// SIMATIC S7-200 SMART project (STEP 7-Micro/WIN SMART), CPU ST20

SYMBOL_TABLE USER1
Btn启动气密          M1.0
Btn停止气密          M1.1
i水箱升到位           M1.2
i水箱j降到位          M1.3
iMaual           M1.4
iAutoGas         M1.5
iResetSingle     M1.6
iStop急停          M1.7
iStartSingle     M2.0
i顶缸上限位           M2.1
i顶杆下限位           M2.2
iHas销钉1          M2.3
iHas销钉2          M2.4
iBYLOK           M2.5
iBYLNG           M2.6
Btn清零合格不合格计数     M2.7
Btn顶缸伸出          M3.0
Btn顶缸缩回          M3.1
Q顶缸伸出启停          M3.2
Q顶缸缩回启停          M3.3
iAutoWater       M3.4
Btn侧顶油伸出         M3.5
Btn侧顶油缩回         M3.6
Q侧顶油伸出启停         M3.7
Q侧顶油缩回启停         M4.0
Btn侧气顶出          M4.2
Btn侧气缩回          M4.3
Q侧气顶出            M4.4
Q侧气缩回            M4.5
Btn高压气检启停        M4.7
Btn低压气检启停        M5.0
Q高压气检启停          M5.1
Q低压气检启停          M5.2
Btn打点伸出          M5.4
Btn打点缩回          M5.5
Q打点伸出            M5.6
Q打点缩回            M5.7
Btn水箱上升启停        M6.1
Btn水箱下降启停        M6.2
Q水箱上升启停          M6.3
Q水箱下降启停          M6.4
Btn高压水检启停        M6.6
Q高压水检启停          M6.7
Btn低压水检启停        M7.0
Q低压水检启停          M7.1
i光栅              M7.3
Btn工作台退回         M7.4
Q工作台推出           M7.5
Q工作台退回           M7.6
Q启动气密仪           M7.7
Q停止气密仪           M8.0
QOK              M8.1
QNG              M8.2
QError报警         M8.3
Q启动运行灯           M8.4
Q三色绿运行           M8.5
Q三色红故障           M8.6
Q三色黄等待           M8.7
Q24V照明灯          M9.0
Q原位指示            M9.1
UISetEnable侧油    M9.3
UISetEnable侧气    M9.4
UISetEnable水箱    M9.5
UISetEnable高压水气检 M9.6
UISetEnable低压水气检 M9.7
UISetEnablee一切换二路 M10.0
MaualVirtual启停气密仪 M10.1
UISetEnable1     M10.2
UIBtnExecute1    M10.3
UISinaPosDone1   M10.4
UISetEnable2     M10.5
UIBtnExecute2    M10.6
UISinaPosDone2   M10.7
UISetEnable销钉    M11.0
CondTrue水箱上升     M11.1
CondTrue水箱下降     M11.2
CondTrue打点伸      M11.3
CondTrue打点缩      M11.4
CondTrueJOG启动气密  M11.5
CondTrueJOG停止气密  M11.6
CondTrue侧气伸      M11.7
CondTrue侧气缩      M12.0
CondTrue一路水检     M12.1
CondTrue二路水检     M12.2
CondTrue有码       M12.3
CondTrue气检合格     M12.4
CondTrue气检不合格    M12.5
CondTrue水检合格     M12.6
CondTrue水检不合格    M12.7
CondTrue工作台推出    M13.0
CondTrue工作台缩回    M13.1
CondTrue顶缸伸      M13.2
CondTrue顶缸缩      M13.3
CondTrue侧油伸      M13.4
CondTrue侧油缩      M13.5
CondTrue一路气检启停   M13.6
CondTrue二路气检启停   M13.7
CondTrue启停气密仪    M14.0
Device当前气密仪状态    M14.1
CondTrue三路气检启停   M14.2
CondTrue关机       M14.3
CondTrueUI气检采集   M14.4
CondTrueUI水检采集   M14.5
UISetEnable扫码枪   M14.6
UIWarning警告      M14.7
UISetSwitch福田    M15.0
CondTrue自锁延迟     M15.1
QLogic伺服启动1      M15.2
QLogic伺服启动2      M15.3
CondTrue伺服启动1    M15.4
CondTrue伺服启动2    M15.5
UIBtnDog上升1      M15.6
UIBtnDog下降1      M15.7
IError泵1         M16.0
IError泵2         M16.1
RunSeq           VW22
UIRunMode        VW28
CountGasRun合格    VW100
CountGasRun不合格   VW102
CountGasRun总数    VW104
RTU扭力1           VW106
RTU扭力2           VW108
UISet无操作待机       VW116
sys待机分钟          VW118
UISet延时复位        VW120
Logic延时复位计时      VW122
UISet福田延时检测      VW124
Logic福田延时计数      VW126
UISetNG福田延时检测    VW128
LogicNG福田延时计数    VW130
UIConv扭力1        VD132
UIConv扭力2        VD136
UISet扭力OK下限1     VD140
UISet扭力OK上限1     VD144
UISet扭力OK下限2     VD148
UISet扭力OK上限2     VD152
UISet伺服距离OK下限1   VD156
UISet伺服距离OK上限1   VD160
UISet伺服距离OK下限2   VD164
UISet伺服距离OK上限2   VD168
UIData扫码枪数据1     VW180
UIData扫码枪数据2     VW182
UIData扫码枪数据3     VW184
UIData扫码枪数据4     VW186
UIData扫码枪数据5     VW188
UIData扫码枪数据6     VW190
UIData扫码枪数据7     VW192
UIData扫码枪数据8     VW194
UIData扫码枪数据9     VW196
UIData扫码枪数据10    VW198
UIData扫码枪数据11    VW200
UIData扫码枪数据12    VW202
UIData扫码枪数据13    VW204
UIData扫码枪数据14    VW206
UIData扫码枪数据15    VW208
UIData扫码枪数据16    VW210
UIData扫码枪数据17    VW212
UIData扫码枪数据18    VW214
UIData扫码枪数据19    VW216
UIData扫码枪数据20    VW218
UIData扫码枪数据21    VW220
UIData扫码枪数据22    VW222
UIData扫码枪数据23    VW224
UIData扫码枪数据24    VW226
UIData扫码枪数据25    VW228
UIData扫码枪数据26    VW230
UIData扫码枪数据27    VW232
UIData扫码枪数据28    VW234
UIData扫码枪数据29    VW236
UIData扫码枪数据30    VW238
UIData扫码枪数据31    VW240
UIData扫码枪数据32    VW242
UIData扫码枪数据33    VW244
UIData扫码枪数据34    VW246
UIData扫码枪数据35    VW248
UIData扫码枪数据36    VW250
UIData扫码枪数据37    VW252
UIData扫码枪数据38    VW254
UIData扫码枪数据39    VW256
UIData扫码枪数据40    VW258
Map气检合格不合格       VW260
UI操作员1           VW262
UI操作员2           VW264
UI操作员3           VW266
UI操作员4           VW268
UI操作员5           VW270
UI操作员6           VW272
UI操作员7           VW274
UI操作员8           VW276
UI操作员9           VW278
UI操作员10          VW280
UI压力值1           VD282
UI扭压力判定结果1       VW286
UI伸出距离1          VD288
UI伸出距离判定1        VW292
UI压力值2           VD294
UI扭压力判定结果2       VW298
UI伸出距离2          VD300
UI伸出距离判定2        VW304
UISetServeMode1  VW500
UISetServePos1   VD502
UISetMDI1        VD506
UISetServeMode2  VW510
UISetServePos2   VD512
UISetMDI2        VD516
UISetZeroOffset1 VD520
UISetZeroOffset2 VD524
Positive1        V600.0
Negative1        V600.1
UISetJodForward1 V600.2
UISetJodReserve1 V600.3
UIBtnFlyRef1     V600.4   // 其他模式下回零
UISetResetErr1   V600.5
UISetOverV1      VW602    // 速度倍率（控制旋转快慢）
UISetOverAcc1    VW604    // 加速倍率（控制启动快慢）
UISetOverDec1    VW606    // 减速度倍率（控制停止快慢）
ConfigEpos1      VD608
ActPosition1     VD612
Axisenabled1     V650.0
AxisPosOk1       V650.1
AxisRef1         V650.2
Lockout1         V650.3
AxisWarn1        V650.4
AxisError1       V650.5
Overrange_Error1 V650.6
ErrorID1         VB651
Positive2        V700.0
Negative2        V700.1
UISetJodForward2 V700.2
UISetJodReserve2 V700.3
UIBtnFlyRef2     V700.4
UISetResetErr2   V700.5
UISetOverV2      VW702
UISetOverAcc2    VW704
UISetOverDec2    VW706
ConfigEpos2      VD708
ActPosition2     VD712
AxisPosOk2       V750.0
AxisRef2         V750.1
Lockout2         V750.2
AxisWarn2        V750.3
AxisError2       V750.4
Overrange_Error2 V750.5
ErrorID2         VB751
LogicMax压力1      VD800
LogicMax压力2      VD804
LogicMax伸出距离1    VD808
LogicMax伸出距离2    VD812
Logic伸出距离1       VD816
Logic伸出距离2       VD820
END_SYMBOL_TABLE

SYMBOL_TABLE 系统符号
Always_On        SM0.0    // 始终接通
First_Scan_On    SM0.1    // 仅在第一个扫描周期时接通
Clock_1s         SM0.5    // 针对 1 s 的周期时间，时钟脉冲接通 0.5 s，断开 0.5 s.
END_SYMBOL_TABLE

SYMBOL_TABLE VarＴ
占1               T37
占2               T38
占3               T39
占4               T40
占5               T41
占6               T42
占7               T43
占8               T44
占9               T45
占10              T46
占11              T47
占12              T48
占13              T49
占14              T50
占15              T51
占16              T52
占17              T53
占18              T54
占19              T55
占20              T56
占21              T57
占22              T58
占23              T59
占24              T60
占25              T61
占26              T62
占27              T63
占28              T101
END_SYMBOL_TABLE

ORGANIZATION_BLOCK MAIN:OB1
TITLE=子程序注释
BEGIN
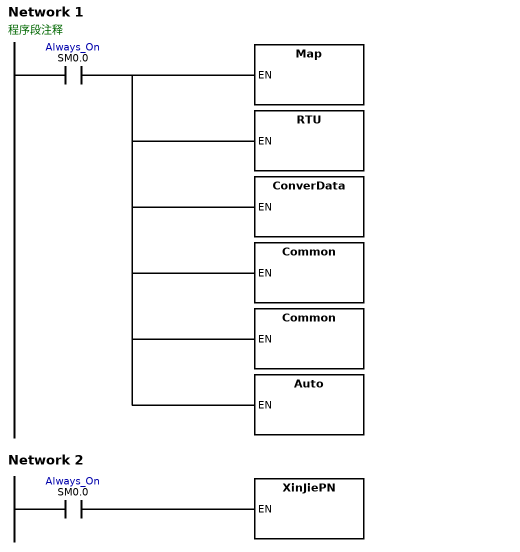
Network 1
// 程序段注释
LD     Always_On:SM0.0
CALL   Map:SBR5
CALL   RTU:SBR4
CALL   ConverData:SBR6
CALL   Common:SBR0
CALL   Common:SBR0
CALL   Auto:SBR3
Network 2
LD     Always_On:SM0.0
CALL   XinJiePN:SBR9
END_ORGANIZATION_BLOCK

SUBROUTINE_BLOCK Common:SBR0
TITLE= 
// SUBROUTINE COMMENTS
// Press F1 for help and example program
//  
VAR
tmpIsRuningGas:BOOL;	// L0.0 
tmpIsWaitGas:BOOL;	// L0.1 
tmpIsRuningWater:BOOL;	// L0.2 
tmpIsWaitWater:BOOL;	// L0.3 
END_VAR
BEGIN
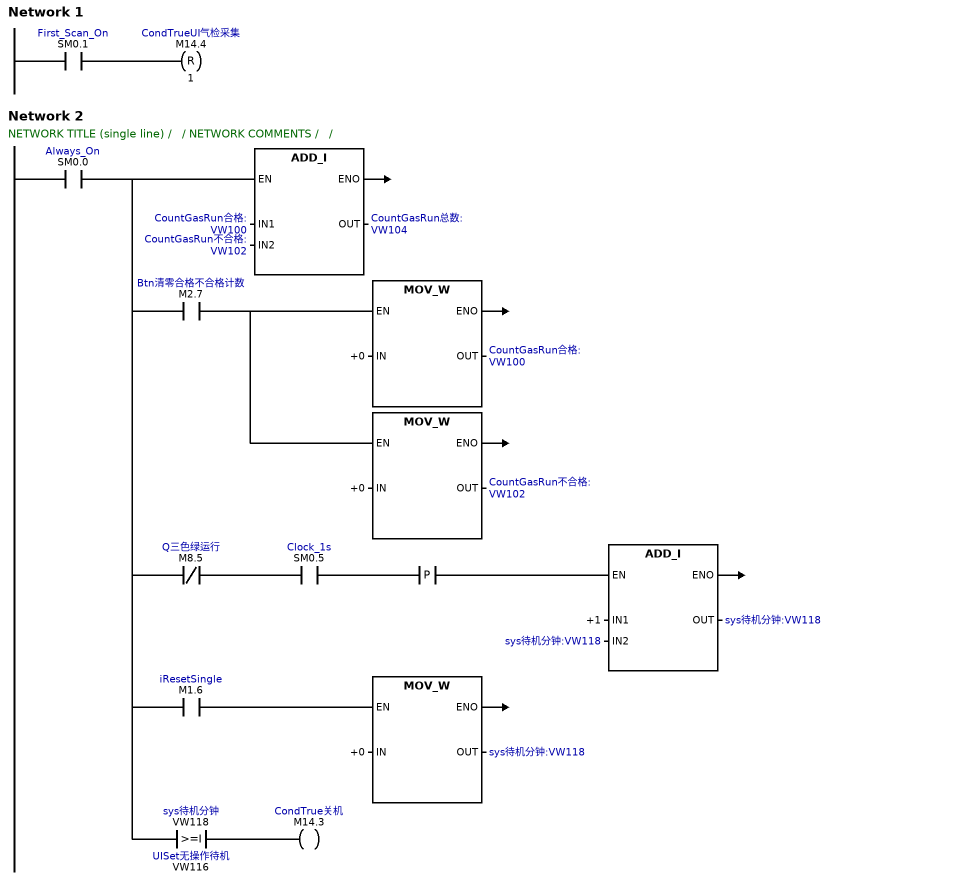
Network 1
LD     First_Scan_On:SM0.1
R      CondTrueUI气检采集:M14.4, 1
Network 2
// NETWORK TITLE (single line)
//  
// NETWORK COMMENTS
//  
// 
LD     Always_On:SM0.0
LPS
MOVW   CountGasRun合格:VW100, CountGasRun总数:VW104
+I     CountGasRun不合格:VW102, CountGasRun总数:VW104
A      Btn清零合格不合格计数:M2.7
MOVW   +0, CountGasRun合格:VW100
MOVW   +0, CountGasRun不合格:VW102
LPP
LPS
AN     Q三色绿运行:M8.5
A      Clock_1s:SM0.5
EU
+I     +1, sys待机分钟:VW118
LRD
A      iResetSingle:M1.6
MOVW   +0, sys待机分钟:VW118
LPP
AW>=   sys待机分钟:VW118, UISet无操作待机:VW116
=      CondTrue关机:M14.3
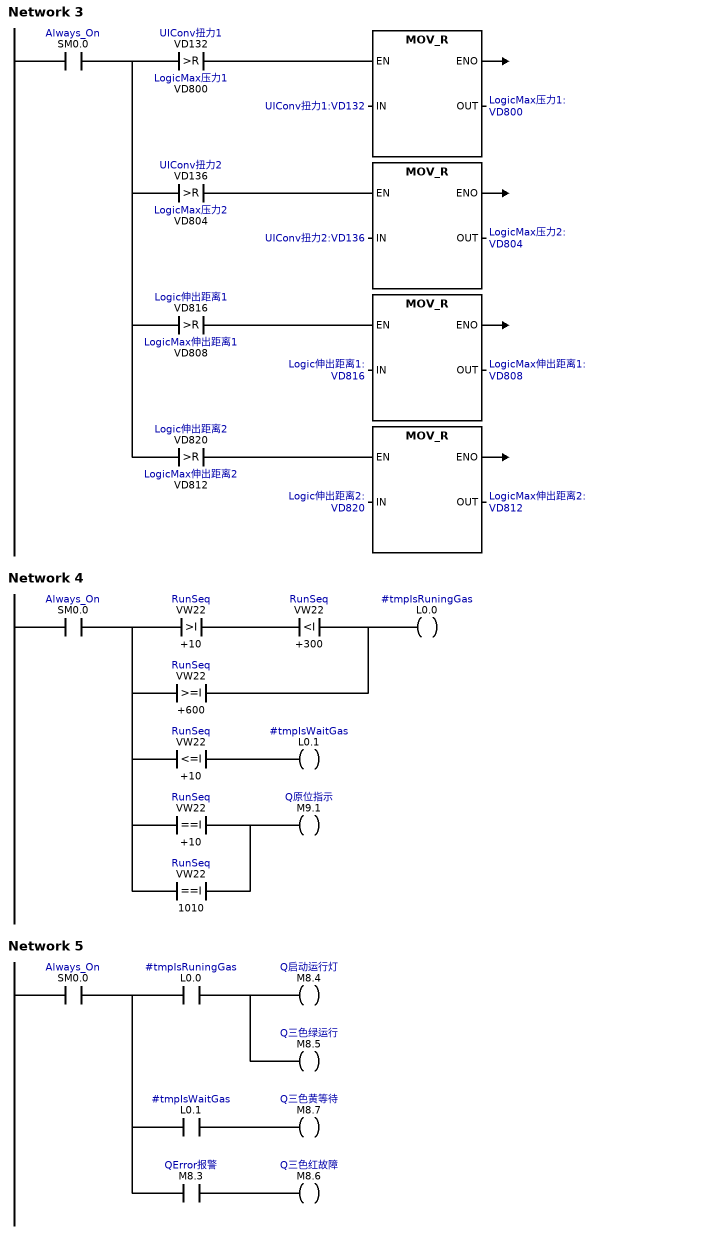
Network 3
LD     Always_On:SM0.0
LPS
AR>    UIConv扭力1:VD132, LogicMax压力1:VD800
MOVR   UIConv扭力1:VD132, LogicMax压力1:VD800
LRD
AR>    UIConv扭力2:VD136, LogicMax压力2:VD804
MOVR   UIConv扭力2:VD136, LogicMax压力2:VD804
LRD
AR>    Logic伸出距离1:VD816, LogicMax伸出距离1:VD808
MOVR   Logic伸出距离1:VD816, LogicMax伸出距离1:VD808
LPP
AR>    Logic伸出距离2:VD820, LogicMax伸出距离2:VD812
MOVR   Logic伸出距离2:VD820, LogicMax伸出距离2:VD812
Network 4
LD     Always_On:SM0.0
LPS
LDW>   RunSeq:VW22, +10
AW<    RunSeq:VW22, +300
OW>=   RunSeq:VW22, +600
ALD
=      #tmpIsRuningGas:L0.0
LRD
AW<=   RunSeq:VW22, +10
=      #tmpIsWaitGas:L0.1
LPP
LDW=   RunSeq:VW22, +10
OW=    RunSeq:VW22, 1010
ALD
=      Q原位指示:M9.1
Network 5
LD     Always_On:SM0.0
LPS
A      #tmpIsRuningGas:L0.0
=      Q启动运行灯:M8.4
=      Q三色绿运行:M8.5
LPP
LPS
A      #tmpIsWaitGas:L0.1
=      Q三色黄等待:M8.7
LPP
A      QError报警:M8.3
=      Q三色红故障:M8.6
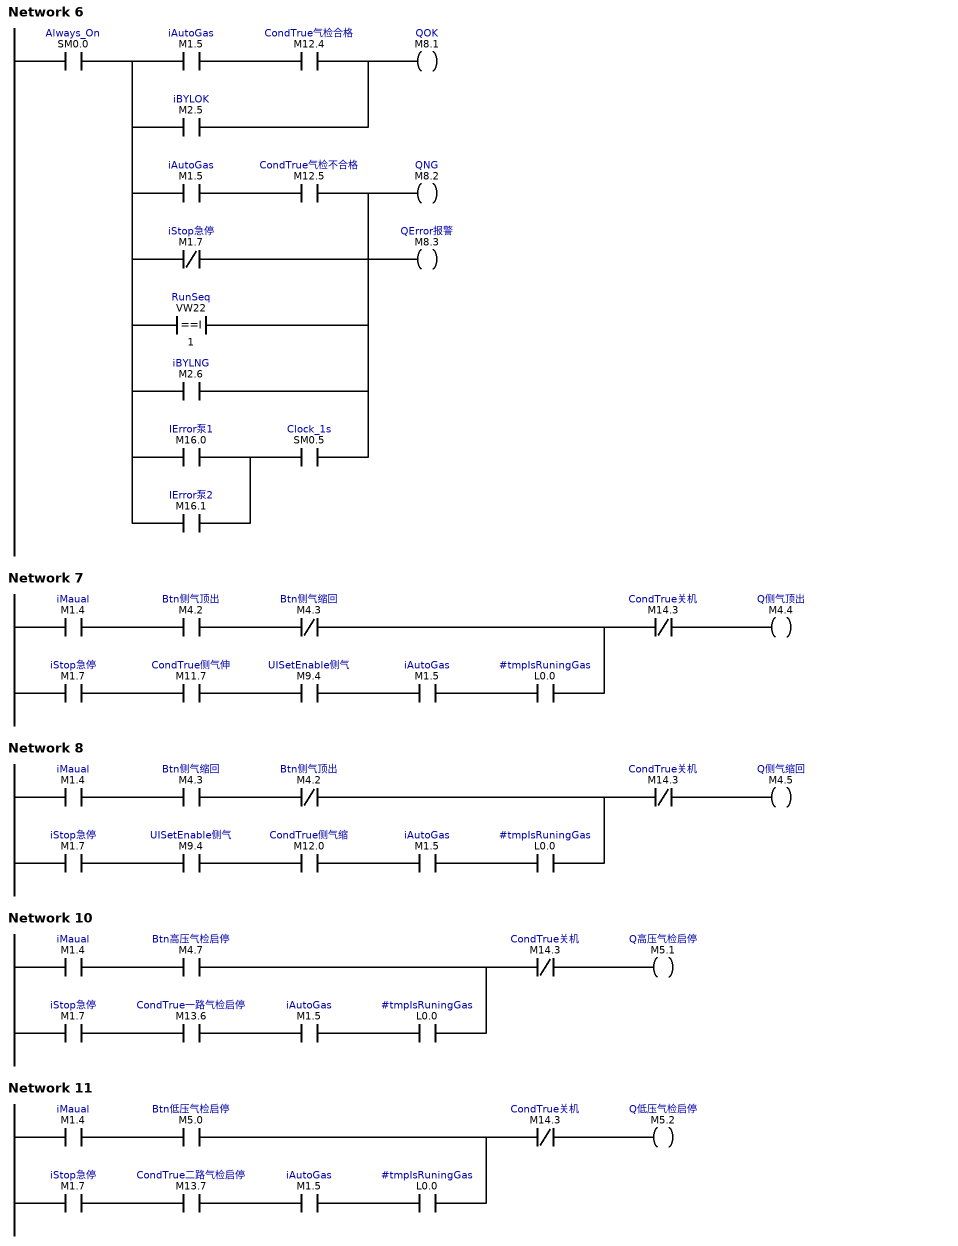
Network 6
LD     Always_On:SM0.0
LPS
LD     iAutoGas:M1.5
A      CondTrue气检合格:M12.4
O      iBYLOK:M2.5
ALD
=      QOK:M8.1
LPP
LD     iAutoGas:M1.5
A      CondTrue气检不合格:M12.5
ON     iStop急停:M1.7
OW=    RunSeq:VW22, 1
O      iBYLNG:M2.6
LD     IError泵1:M16.0
O      IError泵2:M16.1
A      Clock_1s:SM0.5
OLD
ALD
=      QNG:M8.2
=      QError报警:M8.3
Network 7
LD     iMaual:M1.4
A      Btn侧气顶出:M4.2
AN     Btn侧气缩回:M4.3
LD     iStop急停:M1.7
A      CondTrue侧气伸:M11.7
A      UISetEnable侧气:M9.4
A      iAutoGas:M1.5
A      #tmpIsRuningGas:L0.0
OLD
AN     CondTrue关机:M14.3
=      Q侧气顶出:M4.4
Network 8
LD     iMaual:M1.4
A      Btn侧气缩回:M4.3
AN     Btn侧气顶出:M4.2
LD     iStop急停:M1.7
A      UISetEnable侧气:M9.4
A      CondTrue侧气缩:M12.0
A      iAutoGas:M1.5
A      #tmpIsRuningGas:L0.0
OLD
AN     CondTrue关机:M14.3
=      Q侧气缩回:M4.5
Network 10
LD     iMaual:M1.4
A      Btn高压气检启停:M4.7
LD     iStop急停:M1.7
A      CondTrue一路气检启停:M13.6
A      iAutoGas:M1.5
A      #tmpIsRuningGas:L0.0
OLD
AN     CondTrue关机:M14.3
=      Q高压气检启停:M5.1
Network 11
LD     iMaual:M1.4
A      Btn低压气检启停:M5.0
LD     iStop急停:M1.7
A      CondTrue二路气检启停:M13.7
A      iAutoGas:M1.5
A      #tmpIsRuningGas:L0.0
OLD
AN     CondTrue关机:M14.3
=      Q低压气检启停:M5.2
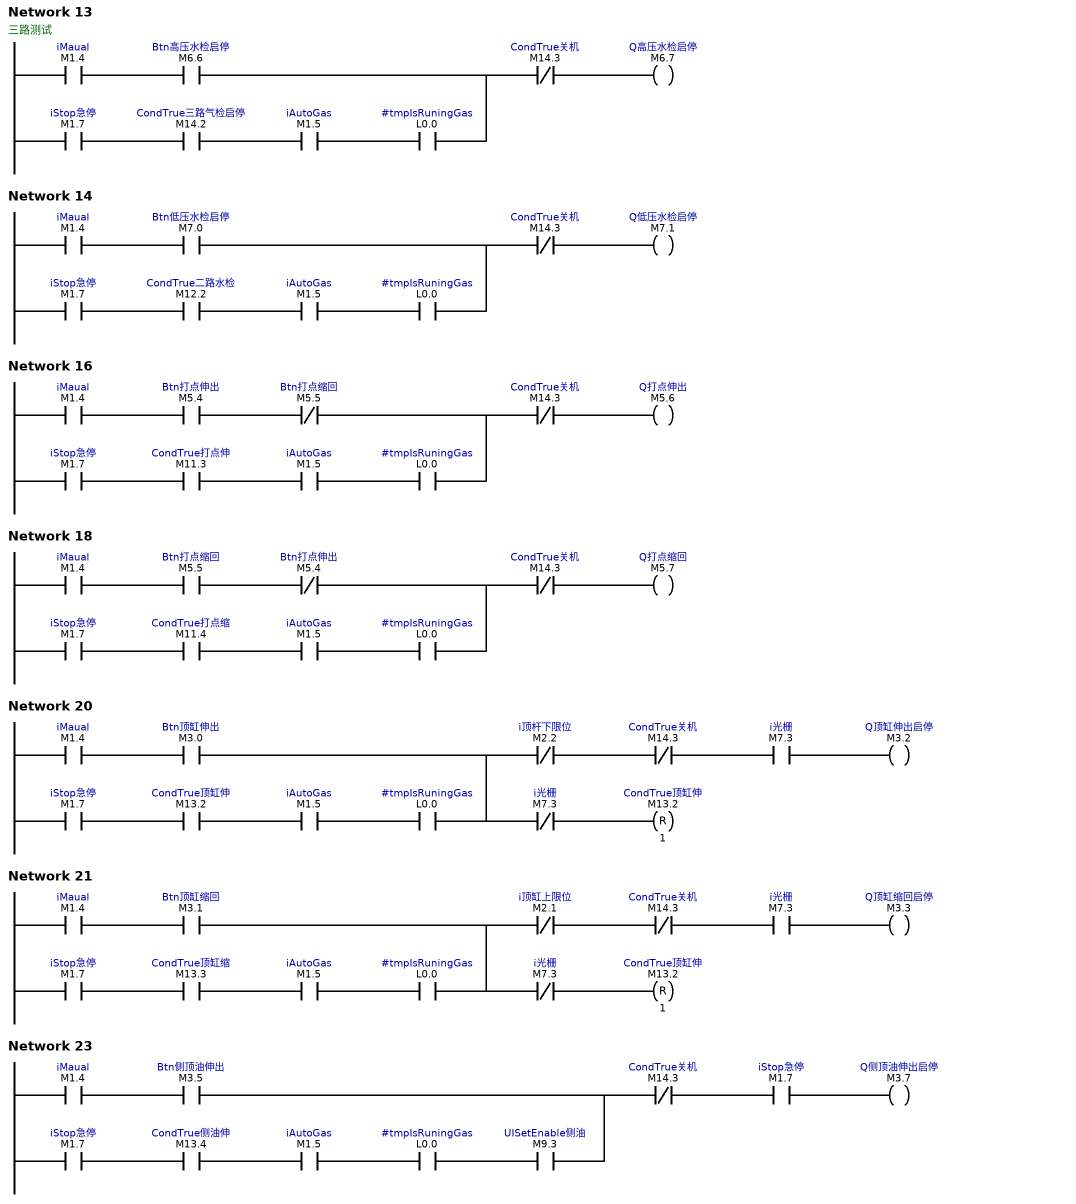
Network 13
// 三路测试
LD     iMaual:M1.4
A      Btn高压水检启停:M6.6
LD     iStop急停:M1.7
A      CondTrue三路气检启停:M14.2
A      iAutoGas:M1.5
A      #tmpIsRuningGas:L0.0
OLD
AN     CondTrue关机:M14.3
=      Q高压水检启停:M6.7
Network 14
LD     iMaual:M1.4
A      Btn低压水检启停:M7.0
LD     iStop急停:M1.7
A      CondTrue二路水检:M12.2
A      iAutoGas:M1.5
A      #tmpIsRuningGas:L0.0
OLD
AN     CondTrue关机:M14.3
=      Q低压水检启停:M7.1
Network 16
LD     iMaual:M1.4
A      Btn打点伸出:M5.4
AN     Btn打点缩回:M5.5
LD     iStop急停:M1.7
A      CondTrue打点伸:M11.3
A      iAutoGas:M1.5
A      #tmpIsRuningGas:L0.0
OLD
AN     CondTrue关机:M14.3
=      Q打点伸出:M5.6
Network 18
LD     iMaual:M1.4
A      Btn打点缩回:M5.5
AN     Btn打点伸出:M5.4
LD     iStop急停:M1.7
A      CondTrue打点缩:M11.4
A      iAutoGas:M1.5
A      #tmpIsRuningGas:L0.0
OLD
AN     CondTrue关机:M14.3
=      Q打点缩回:M5.7
Network 20
LD     iMaual:M1.4
A      Btn顶缸伸出:M3.0
LD     iStop急停:M1.7
A      CondTrue顶缸伸:M13.2
A      iAutoGas:M1.5
A      #tmpIsRuningGas:L0.0
OLD
LPS
AN     i顶杆下限位:M2.2
AN     CondTrue关机:M14.3
A      i光栅:M7.3
=      Q顶缸伸出启停:M3.2
LPP
AN     i光栅:M7.3
R      CondTrue顶缸伸:M13.2, 1
Network 21
LD     iMaual:M1.4
A      Btn顶缸缩回:M3.1
LD     iStop急停:M1.7
A      CondTrue顶缸缩:M13.3
A      iAutoGas:M1.5
A      #tmpIsRuningGas:L0.0
OLD
LPS
AN     i顶缸上限位:M2.1
AN     CondTrue关机:M14.3
A      i光栅:M7.3
=      Q顶缸缩回启停:M3.3
LPP
AN     i光栅:M7.3
R      CondTrue顶缸伸:M13.2, 1
Network 23
LD     iMaual:M1.4
A      Btn侧顶油伸出:M3.5
LD     iStop急停:M1.7
A      CondTrue侧油伸:M13.4
A      iAutoGas:M1.5
A      #tmpIsRuningGas:L0.0
A      UISetEnable侧油:M9.3
OLD
AN     CondTrue关机:M14.3
A      iStop急停:M1.7
=      Q侧顶油伸出启停:M3.7
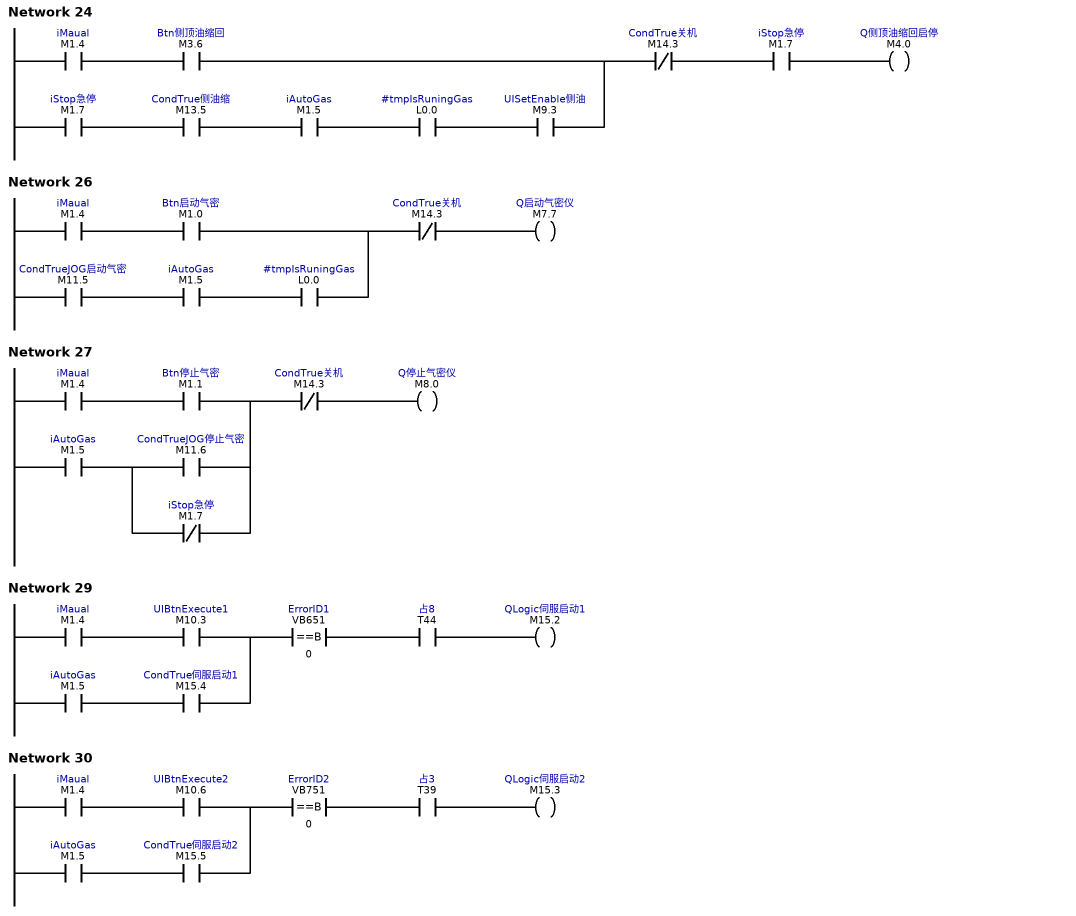
Network 24
LD     iMaual:M1.4
A      Btn侧顶油缩回:M3.6
LD     iStop急停:M1.7
A      CondTrue侧油缩:M13.5
A      iAutoGas:M1.5
A      #tmpIsRuningGas:L0.0
A      UISetEnable侧油:M9.3
OLD
AN     CondTrue关机:M14.3
A      iStop急停:M1.7
=      Q侧顶油缩回启停:M4.0
Network 26
LD     iMaual:M1.4
A      Btn启动气密:M1.0
LD     CondTrueJOG启动气密:M11.5
A      iAutoGas:M1.5
A      #tmpIsRuningGas:L0.0
OLD
AN     CondTrue关机:M14.3
=      Q启动气密仪:M7.7
Network 27
LD     iMaual:M1.4
A      Btn停止气密:M1.1
LD     iAutoGas:M1.5
LD     CondTrueJOG停止气密:M11.6
ON     iStop急停:M1.7
ALD
OLD
AN     CondTrue关机:M14.3
=      Q停止气密仪:M8.0
Network 29
LD     iMaual:M1.4
A      UIBtnExecute1:M10.3
LD     iAutoGas:M1.5
A      CondTrue伺服启动1:M15.4
OLD
AB=    ErrorID1:VB651, 0
A      占8:T44
=      QLogic伺服启动1:M15.2
Network 30
LD     iMaual:M1.4
A      UIBtnExecute2:M10.6
LD     iAutoGas:M1.5
A      CondTrue伺服启动2:M15.5
OLD
AB=    ErrorID2:VB751, 0
A      占3:T39
=      QLogic伺服启动2:M15.3
END_SUBROUTINE_BLOCK

// SBR1: protected block, not included

// SBR2: protected block, not included

SUBROUTINE_BLOCK Auto:SBR3
TITLE=子程序注释
VAR
tmp伺服伸出正误差1:REAL;	// LD0 
tmp伺服伸出负误差1:REAL;	// LD4 
tmp伺服伸出正误差2:REAL;	// LD8 
tmp伺服伸出负误差2:REAL;	// LD12 
END_VAR
BEGIN
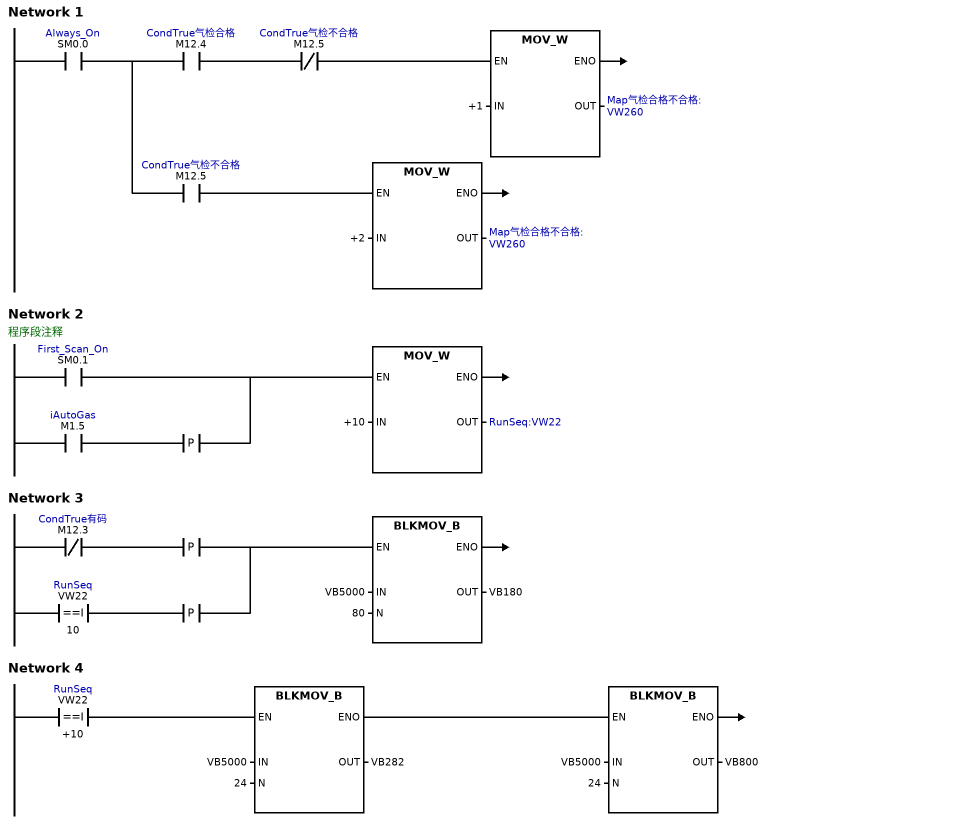
Network 1
LD     Always_On:SM0.0
LPS
A      CondTrue气检合格:M12.4
AN     CondTrue气检不合格:M12.5
MOVW   +1, Map气检合格不合格:VW260
LPP
A      CondTrue气检不合格:M12.5
MOVW   +2, Map气检合格不合格:VW260
Network 2
// 程序段注释
LD     First_Scan_On:SM0.1
LD     iAutoGas:M1.5
EU
OLD
MOVW   +10, RunSeq:VW22
Network 3
LDN    CondTrue有码:M12.3
EU
LDW=   RunSeq:VW22, 10
EU
OLD
BMB    VB5000, VB180, 80
Network 4
LDW=   RunSeq:VW22, +10
BMB    VB5000, VB282, 24
AENO
BMB    VB5000, VB800, 24
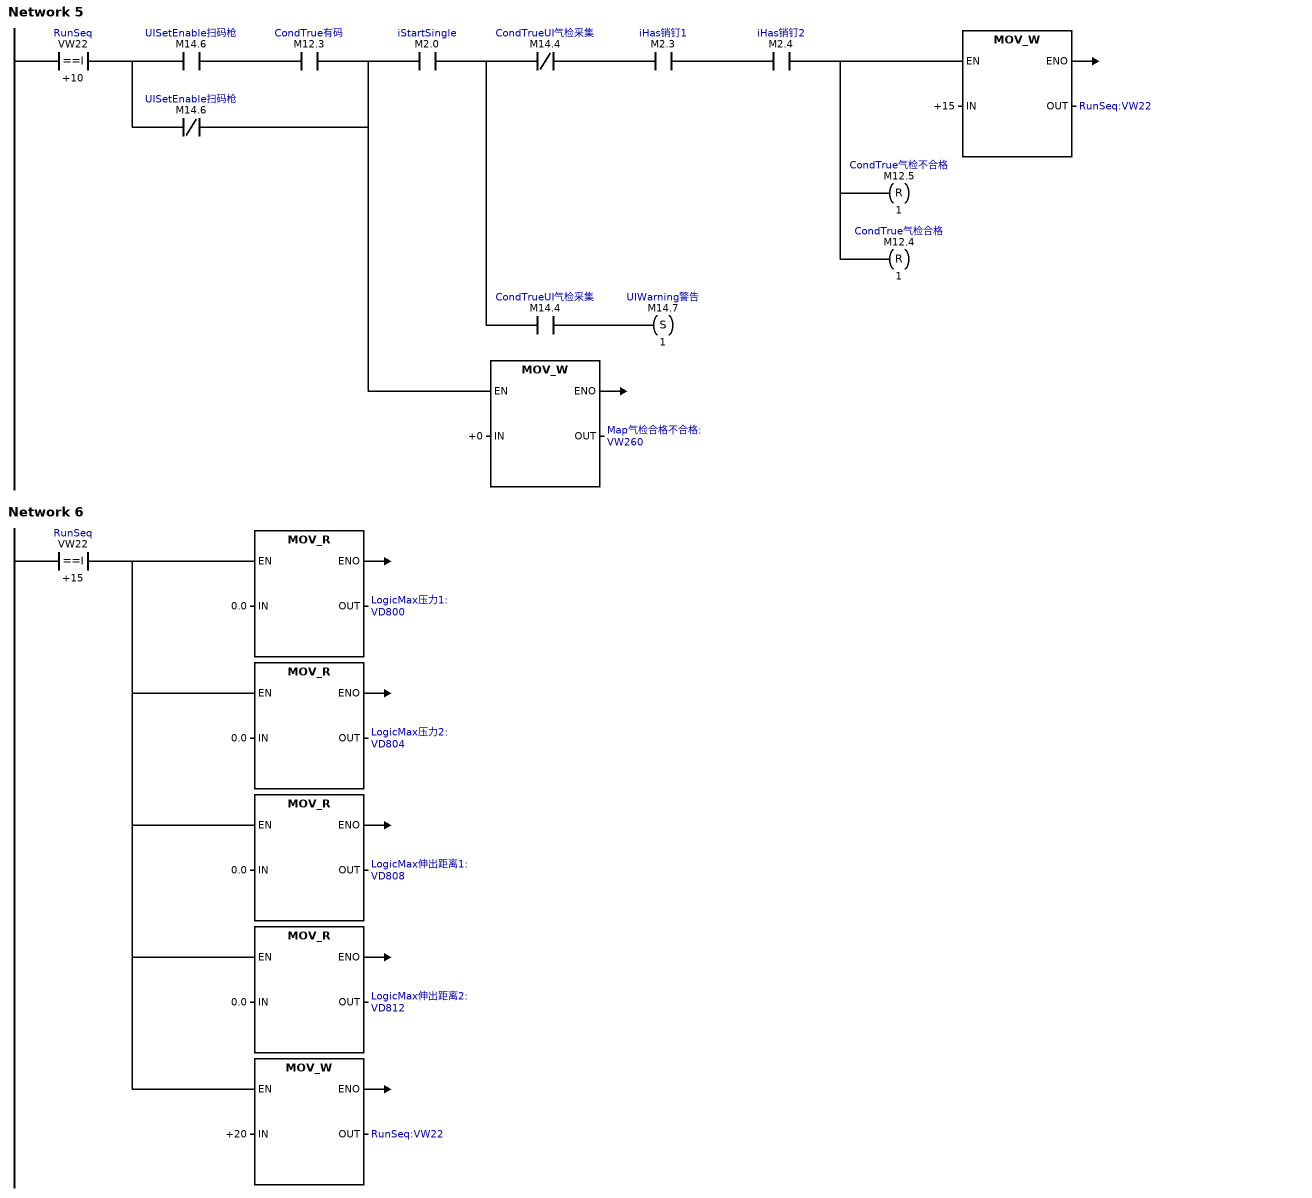
Network 5
LDW=   RunSeq:VW22, +10
LD     UISetEnable扫码枪:M14.6
A      CondTrue有码:M12.3
ON     UISetEnable扫码枪:M14.6
ALD
LPS
A      iStartSingle:M2.0
LPS
AN     CondTrueUI气检采集:M14.4
A      iHas销钉1:M2.3
A      iHas销钉2:M2.4
MOVW   +15, RunSeq:VW22
R      CondTrue气检不合格:M12.5, 1
R      CondTrue气检合格:M12.4, 1
LPP
A      CondTrueUI气检采集:M14.4
S      UIWarning警告:M14.7, 1
LPP
MOVW   +0, Map气检合格不合格:VW260
Network 6
LDW=   RunSeq:VW22, +15
MOVR   0.0, LogicMax压力1:VD800
MOVR   0.0, LogicMax压力2:VD804
MOVR   0.0, LogicMax伸出距离1:VD808
MOVR   0.0, LogicMax伸出距离2:VD812
MOVW   +20, RunSeq:VW22
Network 8
// 1=上限NG
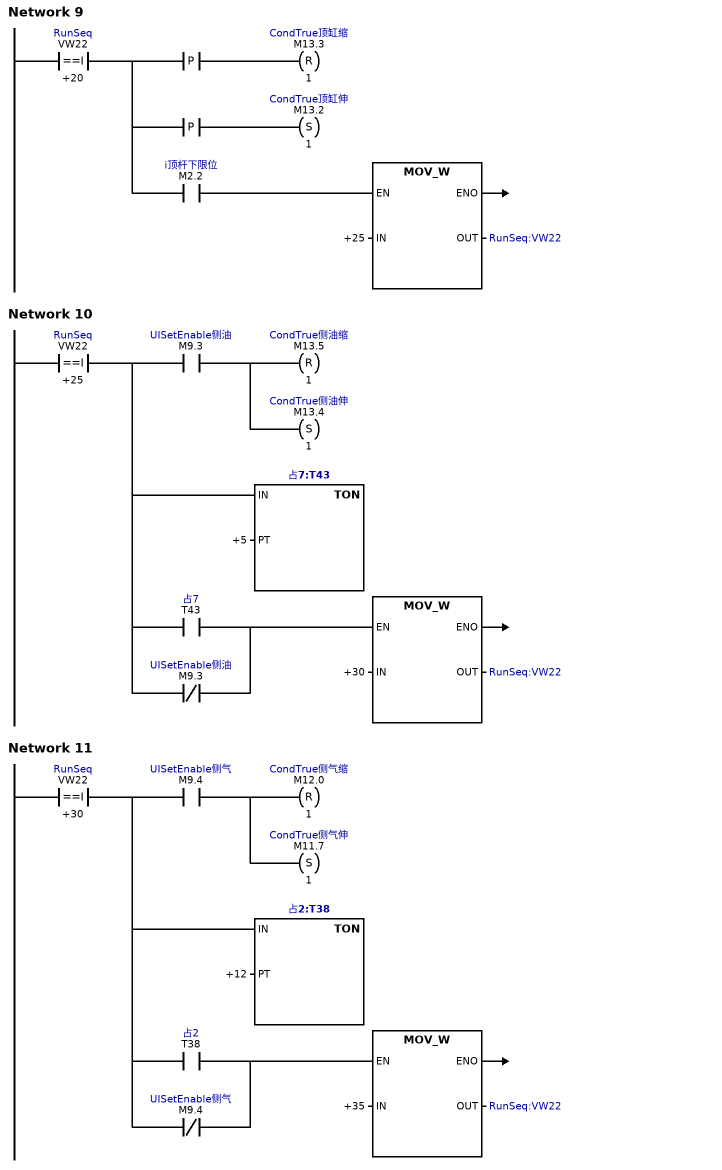
Network 9
LDW=   RunSeq:VW22, +20
LPS
EU
R      CondTrue顶缸缩:M13.3, 1
LRD
EU
S      CondTrue顶缸伸:M13.2, 1
LPP
A      i顶杆下限位:M2.2
MOVW   +25, RunSeq:VW22
Network 10
LDW=   RunSeq:VW22, +25
LPS
A      UISetEnable侧油:M9.3
R      CondTrue侧油缩:M13.5, 1
S      CondTrue侧油伸:M13.4, 1
LRD
TON    占7:T43, +5
LPP
LD     占7:T43
ON     UISetEnable侧油:M9.3
ALD
MOVW   +30, RunSeq:VW22
Network 11
LDW=   RunSeq:VW22, +30
LPS
A      UISetEnable侧气:M9.4
R      CondTrue侧气缩:M12.0, 1
S      CondTrue侧气伸:M11.7, 1
LRD
TON    占2:T38, +12
LPP
LD     占2:T38
ON     UISetEnable侧气:M9.4
ALD
MOVW   +35, RunSeq:VW22
Network 12
// a
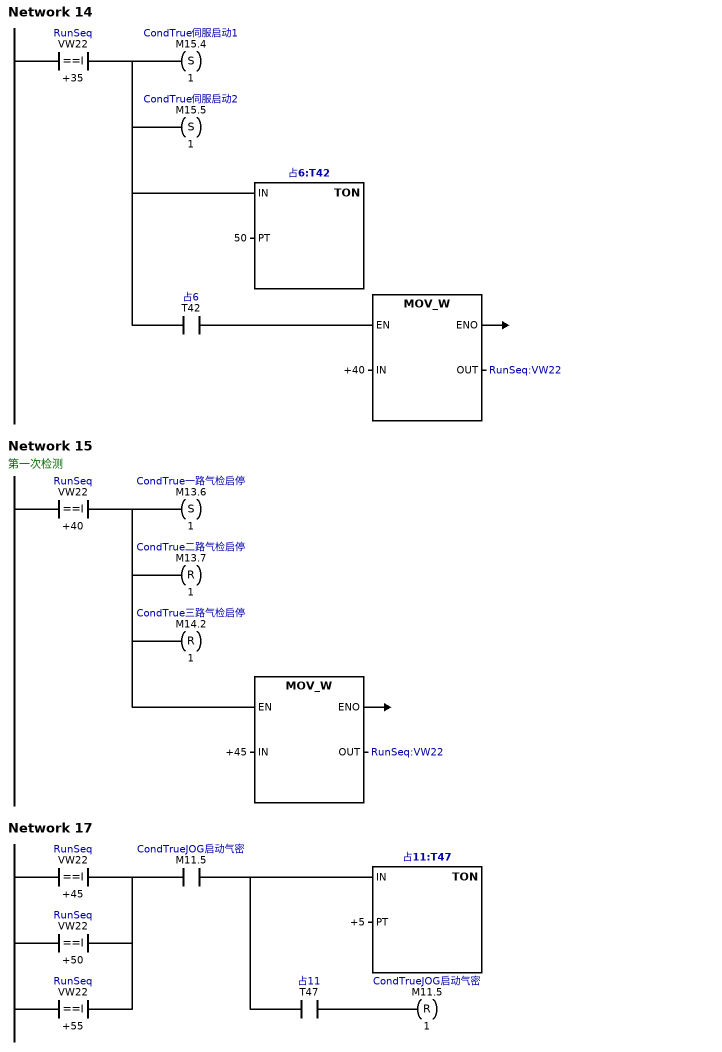
Network 14
LDW=   RunSeq:VW22, +35
S      CondTrue伺服启动1:M15.4, 1
S      CondTrue伺服启动2:M15.5, 1
TON    占6:T42, 50
A      占6:T42
MOVW   +40, RunSeq:VW22
Network 15
// 第一次检测
LDW=   RunSeq:VW22, +40
S      CondTrue一路气检启停:M13.6, 1
R      CondTrue二路气检启停:M13.7, 1
R      CondTrue三路气检启停:M14.2, 1
MOVW   +45, RunSeq:VW22
Network 17
LDW=   RunSeq:VW22, +45
OW=    RunSeq:VW22, +50
OW=    RunSeq:VW22, +55
A      CondTrueJOG启动气密:M11.5
TON    占11:T47, +5
A      占11:T47
R      CondTrueJOG启动气密:M11.5, 1
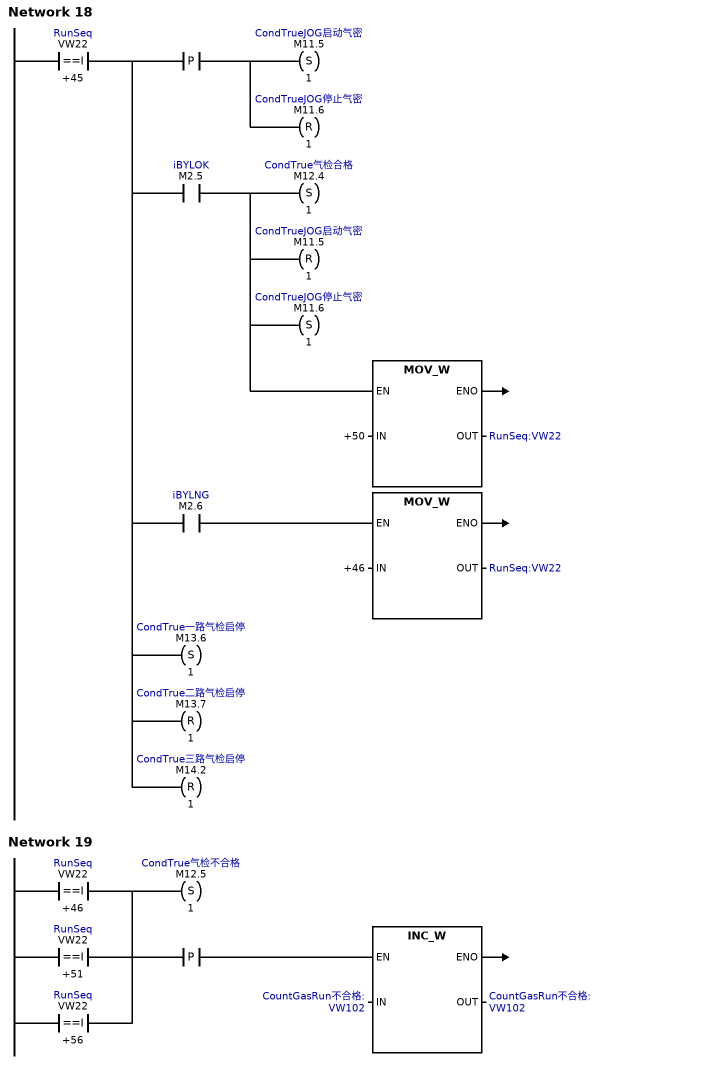
Network 18
LDW=   RunSeq:VW22, +45
LPS
EU
S      CondTrueJOG启动气密:M11.5, 1
R      CondTrueJOG停止气密:M11.6, 1
LRD
A      iBYLOK:M2.5
S      CondTrue气检合格:M12.4, 1
R      CondTrueJOG启动气密:M11.5, 1
S      CondTrueJOG停止气密:M11.6, 1
MOVW   +50, RunSeq:VW22
LPP
LPS
A      iBYLNG:M2.6
MOVW   +46, RunSeq:VW22
LRD
S      CondTrue一路气检启停:M13.6, 1
LRD
R      CondTrue二路气检启停:M13.7, 1
LPP
R      CondTrue三路气检启停:M14.2, 1
Network 19
LDW=   RunSeq:VW22, +46
OW=    RunSeq:VW22, +51
OW=    RunSeq:VW22, +56
S      CondTrue气检不合格:M12.5, 1
EU
INCW   CountGasRun不合格:VW102
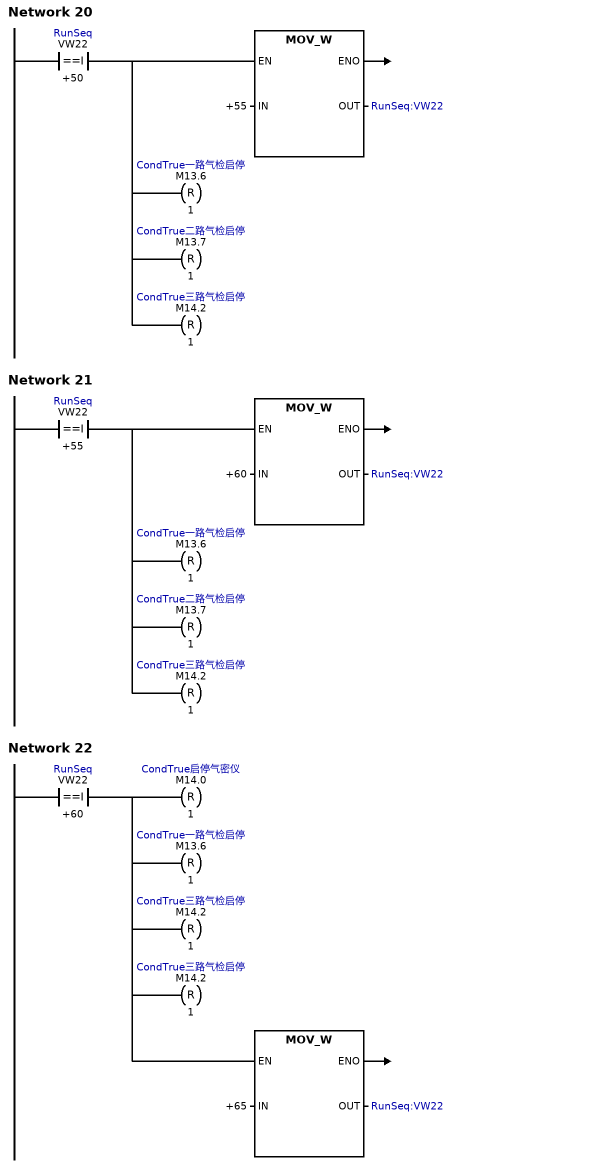
Network 20
LDW=   RunSeq:VW22, +50
MOVW   +55, RunSeq:VW22
R      CondTrue一路气检启停:M13.6, 1
R      CondTrue二路气检启停:M13.7, 1
R      CondTrue三路气检启停:M14.2, 1
Network 21
LDW=   RunSeq:VW22, +55
MOVW   +60, RunSeq:VW22
R      CondTrue一路气检启停:M13.6, 1
R      CondTrue二路气检启停:M13.7, 1
R      CondTrue三路气检启停:M14.2, 1
Network 22
LDW=   RunSeq:VW22, +60
R      CondTrue启停气密仪:M14.0, 1
R      CondTrue一路气检启停:M13.6, 1
R      CondTrue三路气检启停:M14.2, 1
R      CondTrue三路气检启停:M14.2, 1
MOVW   +65, RunSeq:VW22
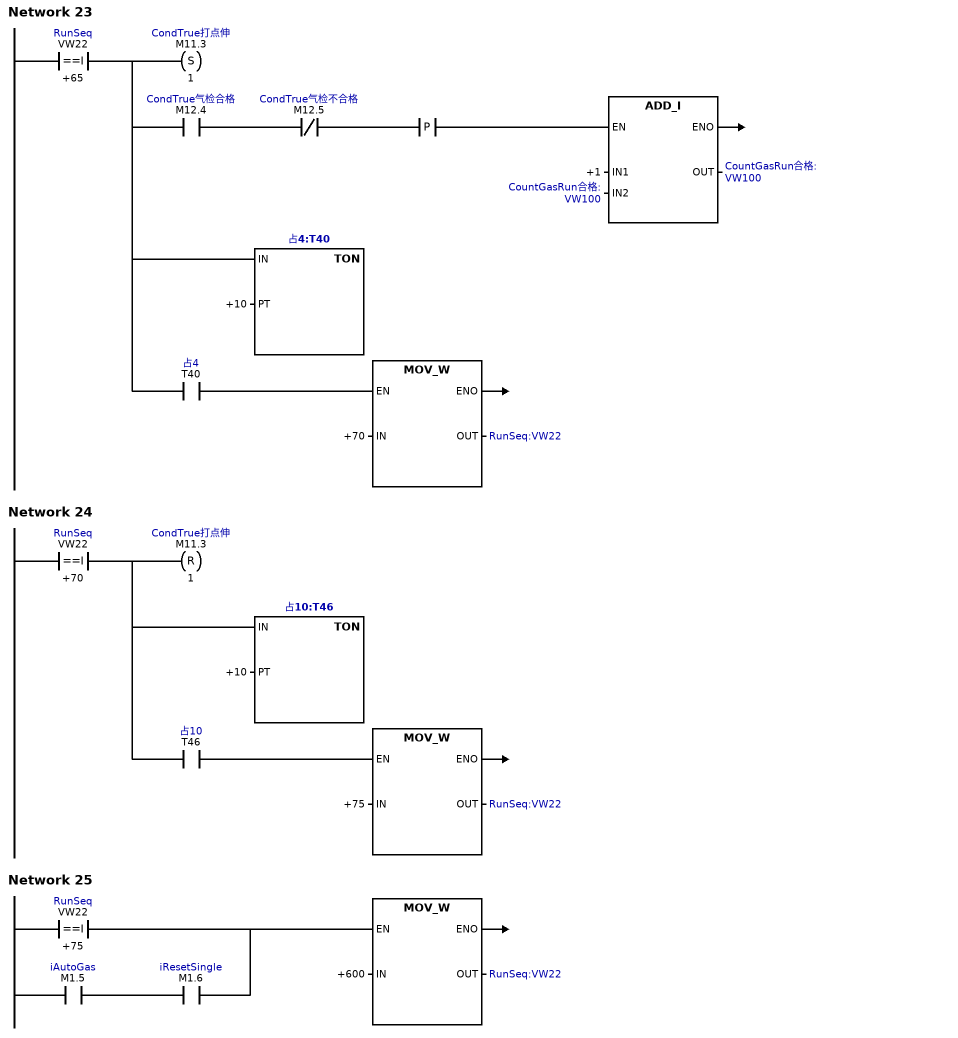
Network 23
LDW=   RunSeq:VW22, +65
LPS
S      CondTrue打点伸:M11.3, 1
A      CondTrue气检合格:M12.4
AN     CondTrue气检不合格:M12.5
EU
+I     +1, CountGasRun合格:VW100
LRD
TON    占4:T40, +10
LPP
A      占4:T40
MOVW   +70, RunSeq:VW22
Network 24
LDW=   RunSeq:VW22, +70
R      CondTrue打点伸:M11.3, 1
TON    占10:T46, +10
A      占10:T46
MOVW   +75, RunSeq:VW22
Network 25
LDW=   RunSeq:VW22, +75
LD     iAutoGas:M1.5
A      iResetSingle:M1.6
OLD
MOVW   +600, RunSeq:VW22
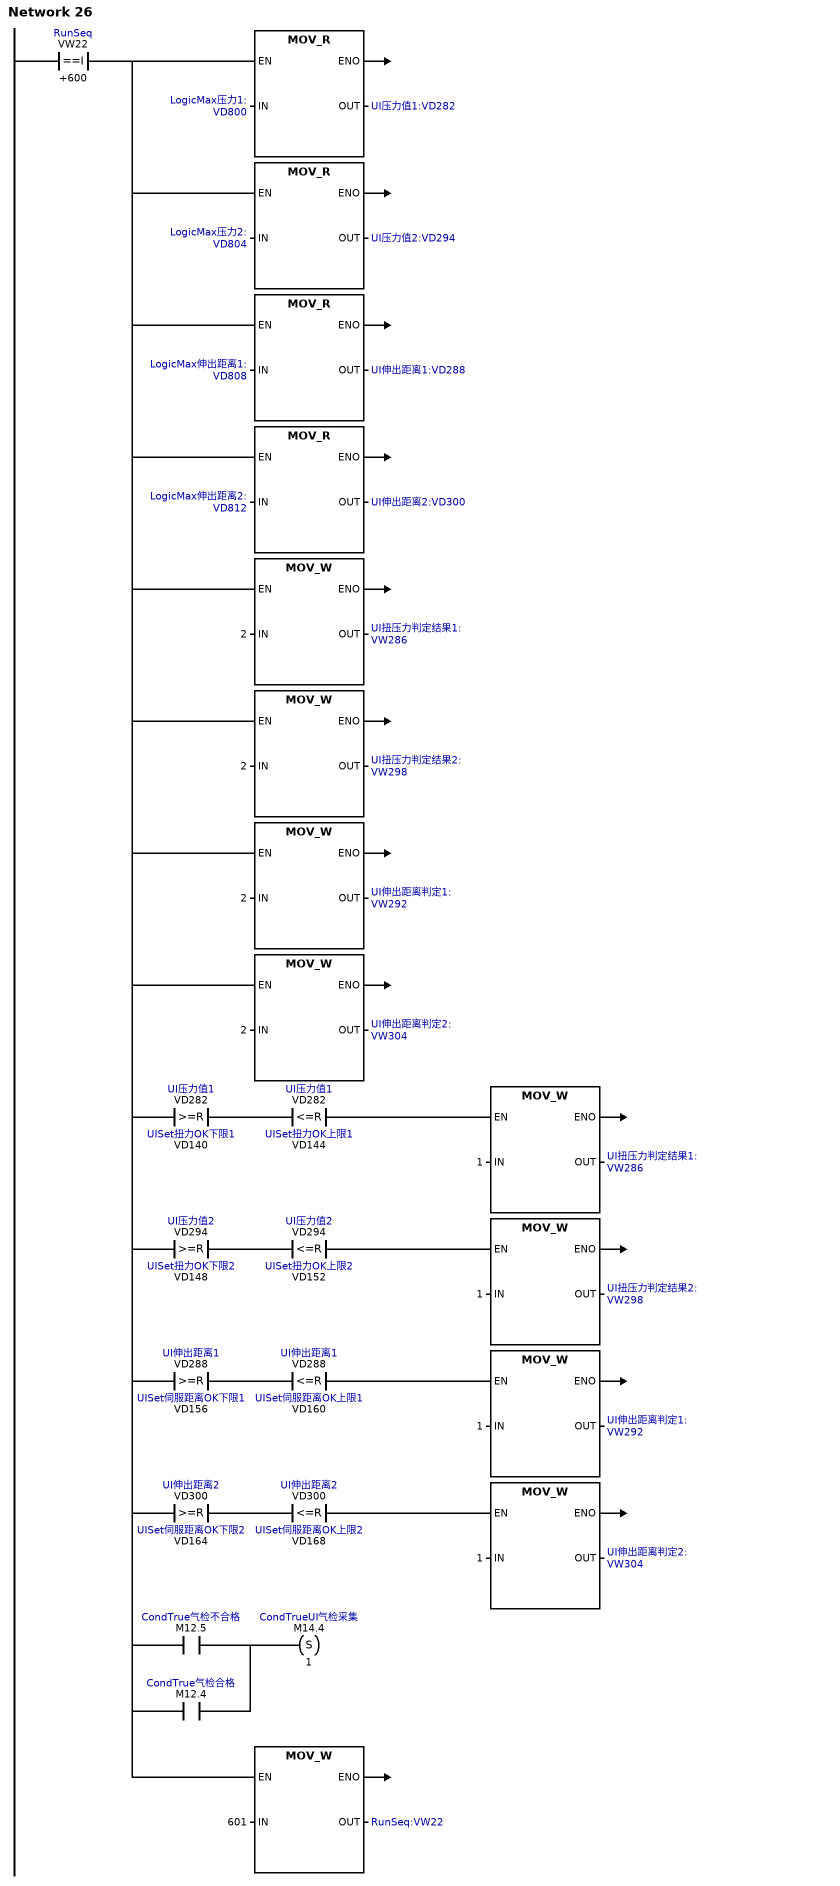
Network 26
LDW=   RunSeq:VW22, +600
LPS
MOVR   LogicMax压力1:VD800, UI压力值1:VD282
MOVR   LogicMax压力2:VD804, UI压力值2:VD294
MOVR   LogicMax伸出距离1:VD808, UI伸出距离1:VD288
MOVR   LogicMax伸出距离2:VD812, UI伸出距离2:VD300
MOVW   2, UI扭压力判定结果1:VW286
MOVW   2, UI扭压力判定结果2:VW298
MOVW   2, UI伸出距离判定1:VW292
MOVW   2, UI伸出距离判定2:VW304
AR>=   UI压力值1:VD282, UISet扭力OK下限1:VD140
AR<=   UI压力值1:VD282, UISet扭力OK上限1:VD144
MOVW   1, UI扭压力判定结果1:VW286
LRD
AR>=   UI压力值2:VD294, UISet扭力OK下限2:VD148
AR<=   UI压力值2:VD294, UISet扭力OK上限2:VD152
MOVW   1, UI扭压力判定结果2:VW298
LRD
AR>=   UI伸出距离1:VD288, UISet伺服距离OK下限1:VD156
AR<=   UI伸出距离1:VD288, UISet伺服距离OK上限1:VD160
MOVW   1, UI伸出距离判定1:VW292
LRD
AR>=   UI伸出距离2:VD300, UISet伺服距离OK下限2:VD164
AR<=   UI伸出距离2:VD300, UISet伺服距离OK上限2:VD168
MOVW   1, UI伸出距离判定2:VW304
LRD
LD     CondTrue气检不合格:M12.5
O      CondTrue气检合格:M12.4
ALD
S      CondTrueUI气检采集:M14.4, 1
LPP
MOVW   601, RunSeq:VW22
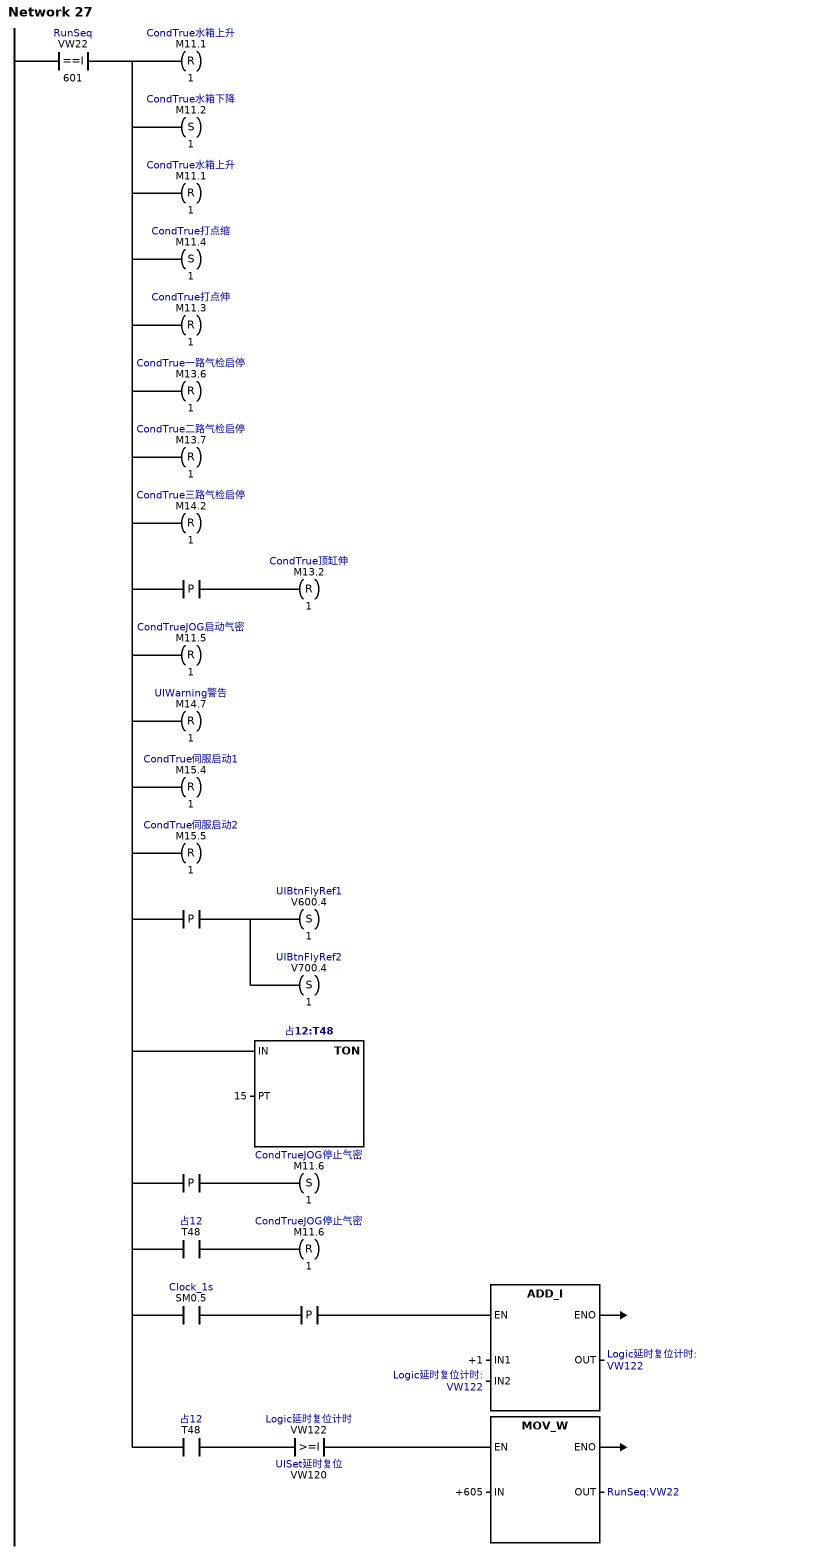
Network 27
LDW=   RunSeq:VW22, 601
LPS
R      CondTrue水箱上升:M11.1, 1
S      CondTrue水箱下降:M11.2, 1
R      CondTrue水箱上升:M11.1, 1
S      CondTrue打点缩:M11.4, 1
R      CondTrue打点伸:M11.3, 1
R      CondTrue一路气检启停:M13.6, 1
R      CondTrue二路气检启停:M13.7, 1
R      CondTrue三路气检启停:M14.2, 1
EU
R      CondTrue顶缸伸:M13.2, 1
LRD
R      CondTrueJOG启动气密:M11.5, 1
LRD
R      UIWarning警告:M14.7, 1
LRD
R      CondTrue伺服启动1:M15.4, 1
LRD
R      CondTrue伺服启动2:M15.5, 1
LRD
EU
S      UIBtnFlyRef1:V600.4, 1
S      UIBtnFlyRef2:V700.4, 1
LPP
LPS
TON    占12:T48, 15
EU
S      CondTrueJOG停止气密:M11.6, 1
LRD
A      占12:T48
R      CondTrueJOG停止气密:M11.6, 1
LRD
A      Clock_1s:SM0.5
EU
+I     +1, Logic延时复位计时:VW122
LPP
A      占12:T48
AW>=   Logic延时复位计时:VW122, UISet延时复位:VW120
MOVW   +605, RunSeq:VW22
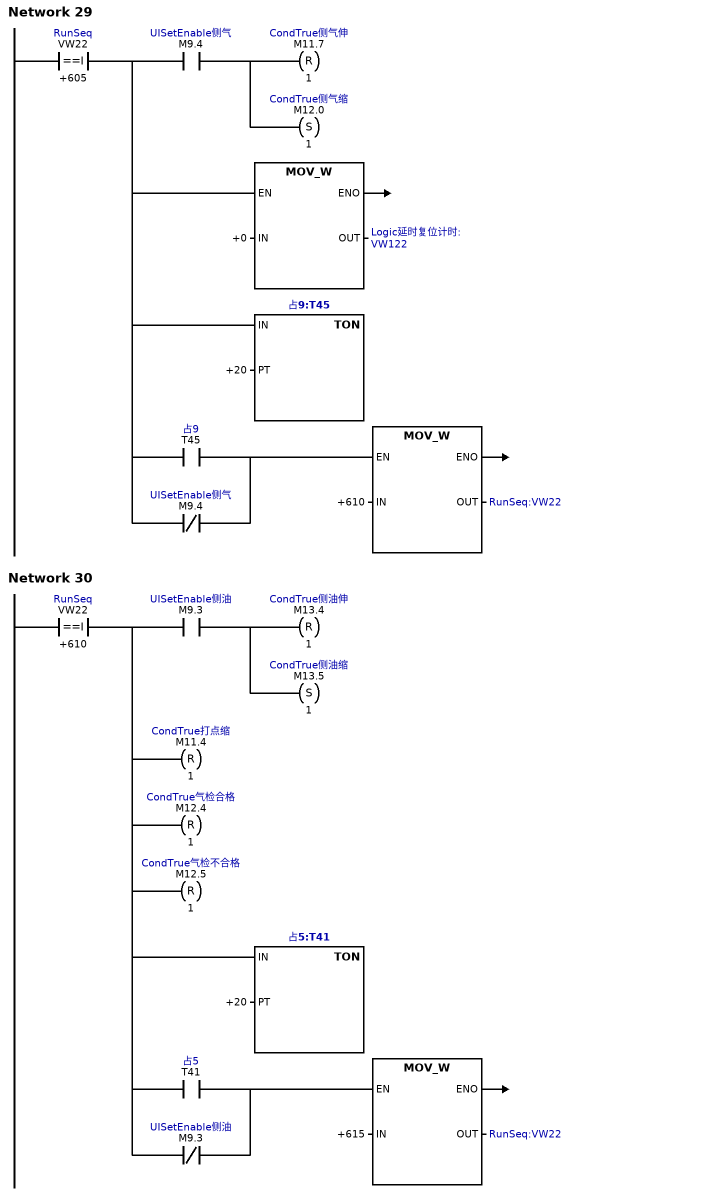
Network 29
LDW=   RunSeq:VW22, +605
LPS
A      UISetEnable侧气:M9.4
R      CondTrue侧气伸:M11.7, 1
S      CondTrue侧气缩:M12.0, 1
LRD
MOVW   +0, Logic延时复位计时:VW122
TON    占9:T45, +20
LPP
LD     占9:T45
ON     UISetEnable侧气:M9.4
ALD
MOVW   +610, RunSeq:VW22
Network 30
LDW=   RunSeq:VW22, +610
LPS
A      UISetEnable侧油:M9.3
R      CondTrue侧油伸:M13.4, 1
S      CondTrue侧油缩:M13.5, 1
LRD
R      CondTrue打点缩:M11.4, 1
R      CondTrue气检合格:M12.4, 1
R      CondTrue气检不合格:M12.5, 1
TON    占5:T41, +20
LPP
LD     占5:T41
ON     UISetEnable侧油:M9.3
ALD
MOVW   +615, RunSeq:VW22
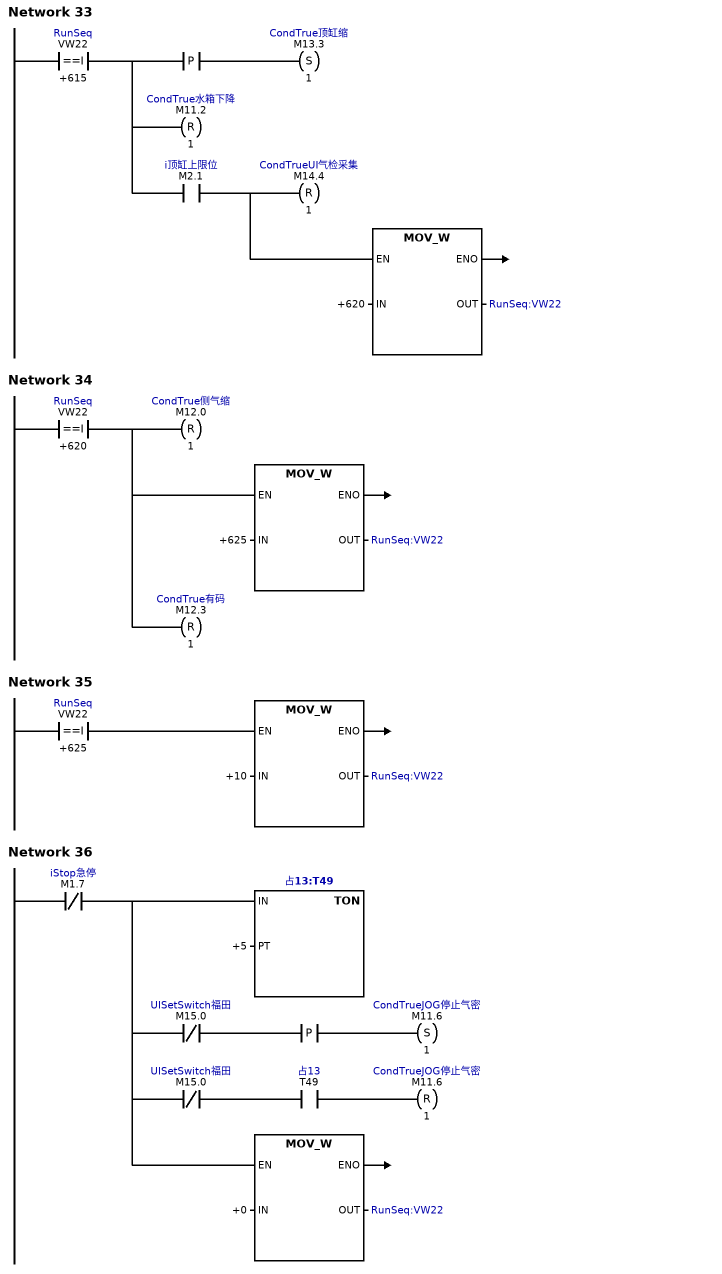
Network 33
LDW=   RunSeq:VW22, +615
LPS
EU
S      CondTrue顶缸缩:M13.3, 1
LRD
R      CondTrue水箱下降:M11.2, 1
LPP
A      i顶缸上限位:M2.1
R      CondTrueUI气检采集:M14.4, 1
MOVW   +620, RunSeq:VW22
Network 34
LDW=   RunSeq:VW22, +620
R      CondTrue侧气缩:M12.0, 1
MOVW   +625, RunSeq:VW22
R      CondTrue有码:M12.3, 1
Network 35
LDW=   RunSeq:VW22, +625
MOVW   +10, RunSeq:VW22
Network 36
LDN    iStop急停:M1.7
LPS
TON    占13:T49, +5
AN     UISetSwitch福田:M15.0
EU
S      CondTrueJOG停止气密:M11.6, 1
LRD
AN     UISetSwitch福田:M15.0
A      占13:T49
R      CondTrueJOG停止气密:M11.6, 1
LPP
MOVW   +0, RunSeq:VW22
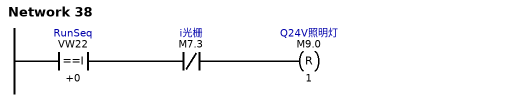
Network 38
LDW=   RunSeq:VW22, +0
AN     i光栅:M7.3
R      Q24V照明灯:M9.0, 1
END_SUBROUTINE_BLOCK

SUBROUTINE_BLOCK RTU:SBR4
TITLE=子程序注释
VAR
tmpDone:BOOL;	// L0.0 
tmpErr:BYTE;	// LB1 
END_VAR
BEGIN
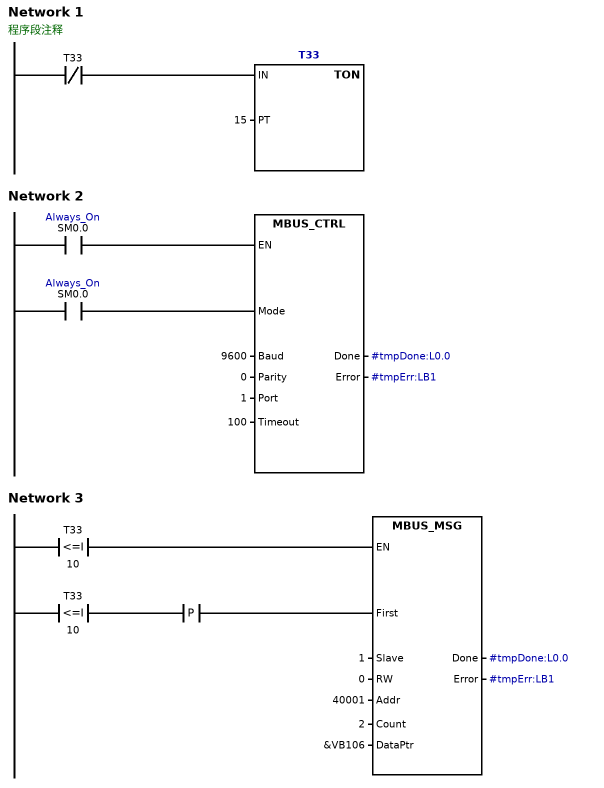
Network 1
// 程序段注释
LDN    T33
TON    T33, 15
Network 2
LD     Always_On:SM0.0
=      L60.0
LD     Always_On:SM0.0
=      L63.7
LD     L60.0
CALL   MBUS_CTRL:SBR10, L63.7, 9600, 0, 1, 100, #tmpDone:L0.0, #tmpErr:LB1
Network 3
LDW<=  T33, 10
=      L60.0
LDW<=  T33, 10
EU
=      L63.7
LD     L60.0
CALL   MBUS_MSG:SBR11, L63.7, 1, 0, 40001, 2, &VB106, #tmpDone:L0.0, #tmpErr:LB1
END_SUBROUTINE_BLOCK

SUBROUTINE_BLOCK Map:SBR5
TITLE=子程序注释
BEGIN
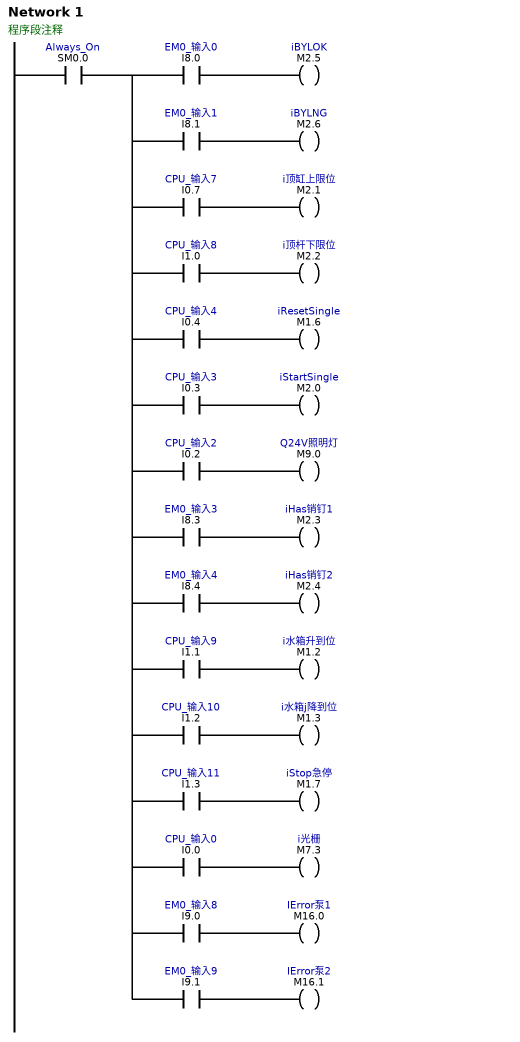
Network 1
// 程序段注释
LD     Always_On:SM0.0
LPS
A      EM0_输入0:I8.0
=      iBYLOK:M2.5
LRD
A      EM0_输入1:I8.1
=      iBYLNG:M2.6
LRD
A      CPU_输入7:I0.7
=      i顶缸上限位:M2.1
LRD
A      CPU_输入8:I1.0
=      i顶杆下限位:M2.2
LRD
A      CPU_输入4:I0.4
=      iResetSingle:M1.6
LRD
A      CPU_输入3:I0.3
=      iStartSingle:M2.0
LRD
A      CPU_输入2:I0.2
=      Q24V照明灯:M9.0
LRD
A      EM0_输入3:I8.3
=      iHas销钉1:M2.3
LRD
A      EM0_输入4:I8.4
=      iHas销钉2:M2.4
LRD
A      CPU_输入9:I1.1
=      i水箱升到位:M1.2
LRD
A      CPU_输入10:I1.2
=      i水箱j降到位:M1.3
LRD
A      CPU_输入11:I1.3
=      iStop急停:M1.7
LRD
A      CPU_输入0:I0.0
=      i光栅:M7.3
LRD
A      EM0_输入8:I9.0
=      IError泵1:M16.0
LPP
A      EM0_输入9:I9.1
=      IError泵2:M16.1
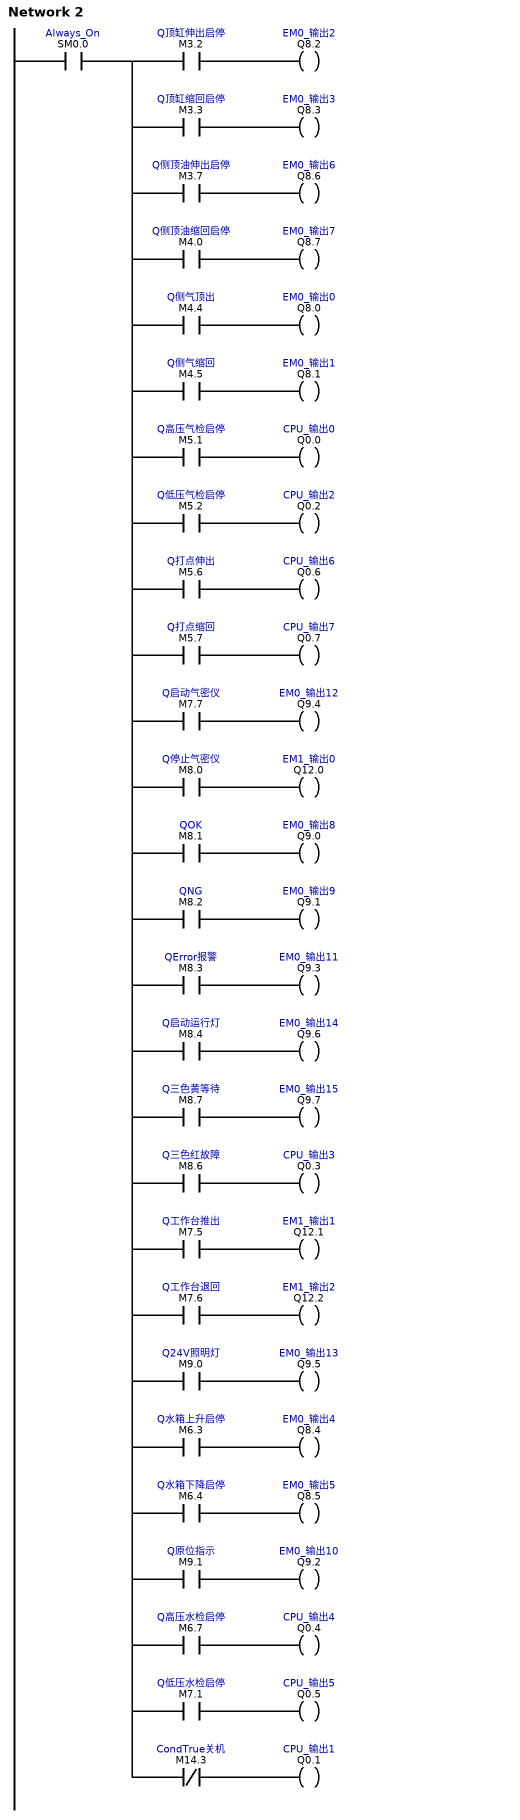
Network 2
LD     Always_On:SM0.0
LPS
A      Q顶缸伸出启停:M3.2
=      EM0_输出2:Q8.2
LRD
A      Q顶缸缩回启停:M3.3
=      EM0_输出3:Q8.3
LRD
A      Q侧顶油伸出启停:M3.7
=      EM0_输出6:Q8.6
LRD
A      Q侧顶油缩回启停:M4.0
=      EM0_输出7:Q8.7
LRD
A      Q侧气顶出:M4.4
=      EM0_输出0:Q8.0
LRD
A      Q侧气缩回:M4.5
=      EM0_输出1:Q8.1
LRD
A      Q高压气检启停:M5.1
=      CPU_输出0:Q0.0
LRD
A      Q低压气检启停:M5.2
=      CPU_输出2:Q0.2
LRD
A      Q打点伸出:M5.6
=      CPU_输出6:Q0.6
LRD
A      Q打点缩回:M5.7
=      CPU_输出7:Q0.7
LRD
A      Q启动气密仪:M7.7
=      EM0_输出12:Q9.4
LRD
A      Q停止气密仪:M8.0
=      EM1_输出0:Q12.0
LRD
A      QOK:M8.1
=      EM0_输出8:Q9.0
LRD
A      QNG:M8.2
=      EM0_输出9:Q9.1
LRD
A      QError报警:M8.3
=      EM0_输出11:Q9.3
LRD
A      Q启动运行灯:M8.4
=      EM0_输出14:Q9.6
LRD
A      Q三色黄等待:M8.7
=      EM0_输出15:Q9.7
LRD
A      Q三色红故障:M8.6
=      CPU_输出3:Q0.3
LRD
A      Q工作台推出:M7.5
=      EM1_输出1:Q12.1
LRD
A      Q工作台退回:M7.6
=      EM1_输出2:Q12.2
LRD
A      Q24V照明灯:M9.0
=      EM0_输出13:Q9.5
LRD
A      Q水箱上升启停:M6.3
=      EM0_输出4:Q8.4
LRD
A      Q水箱下降启停:M6.4
=      EM0_输出5:Q8.5
LRD
A      Q原位指示:M9.1
=      EM0_输出10:Q9.2
LRD
A      Q高压水检启停:M6.7
=      CPU_输出4:Q0.4
LRD
A      Q低压水检启停:M7.1
=      CPU_输出5:Q0.5
LPP
AN     CondTrue关机:M14.3
=      CPU_输出1:Q0.1
END_SUBROUTINE_BLOCK

SUBROUTINE_BLOCK ConverData:SBR6
TITLE=子程序注释
VAR
tmpDint:DINT;	// LD0 
tmpReal:REAL;	// LD4 
END_VAR
BEGIN
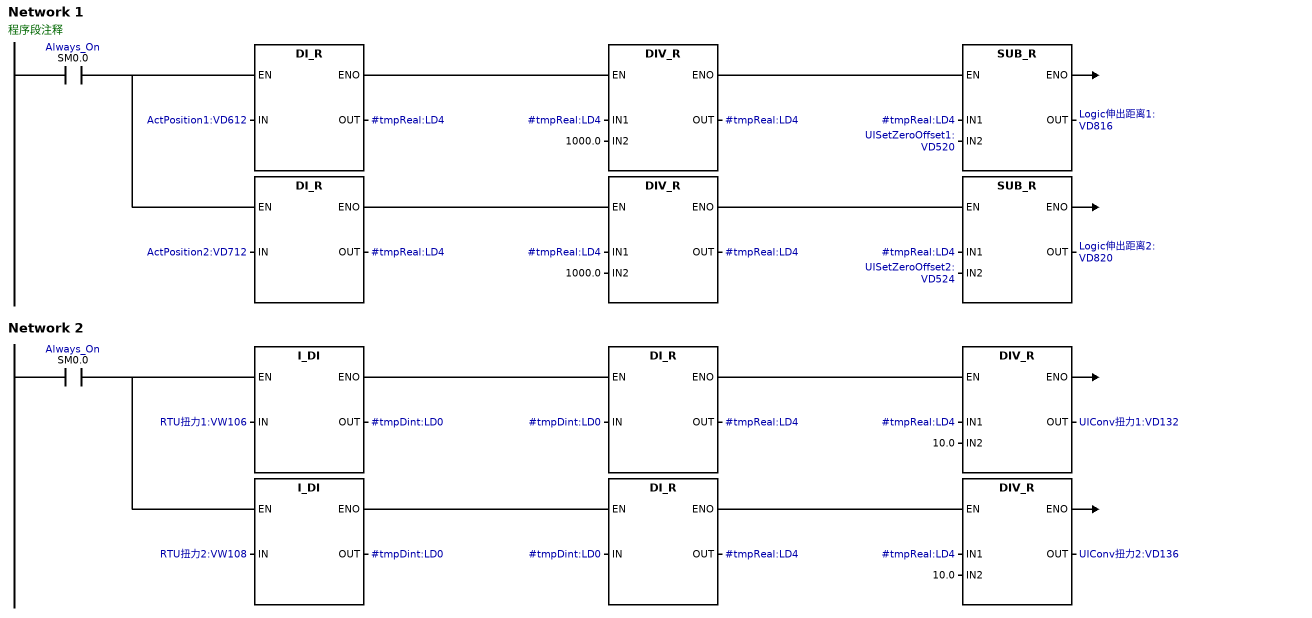
Network 1
// 程序段注释
LD     Always_On:SM0.0
LPS
DTR    ActPosition1:VD612, #tmpReal:LD4
AENO
/R     1000.0, #tmpReal:LD4
AENO
MOVR   #tmpReal:LD4, Logic伸出距离1:VD816
-R     UISetZeroOffset1:VD520, Logic伸出距离1:VD816
LPP
DTR    ActPosition2:VD712, #tmpReal:LD4
AENO
/R     1000.0, #tmpReal:LD4
AENO
MOVR   #tmpReal:LD4, Logic伸出距离2:VD820
-R     UISetZeroOffset2:VD524, Logic伸出距离2:VD820
Network 2
LD     Always_On:SM0.0
LPS
ITD    RTU扭力1:VW106, #tmpDint:LD0
AENO
DTR    #tmpDint:LD0, #tmpReal:LD4
AENO
MOVR   #tmpReal:LD4, UIConv扭力1:VD132
/R     10.0, UIConv扭力1:VD132
LPP
ITD    RTU扭力2:VW108, #tmpDint:LD0
AENO
DTR    #tmpDint:LD0, #tmpReal:LD4
AENO
MOVR   #tmpReal:LD4, UIConv扭力2:VD136
/R     10.0, UIConv扭力2:VD136
END_SUBROUTINE_BLOCK

// SBR7: protected block, not included

// SBR8: protected block, not included

SUBROUTINE_BLOCK XinJiePN:SBR9
TITLE=子程序注释
VAR
tmpSpeed:DWORD;	// LD0 
tmpPos1:DINT;	// LD4 
tmpWarning:WORD;	// LW8 
tmpErr:WORD;	// LW10 
tmpDone:BOOL;	// L12.0 
tmpNotJOD:BOOL;	// L12.1 
tmpPos2:DINT;	// LD13 
tmpReal:REAL;	// LD17 
tmpDint:DINT;	// LD21 
END_VAR
BEGIN
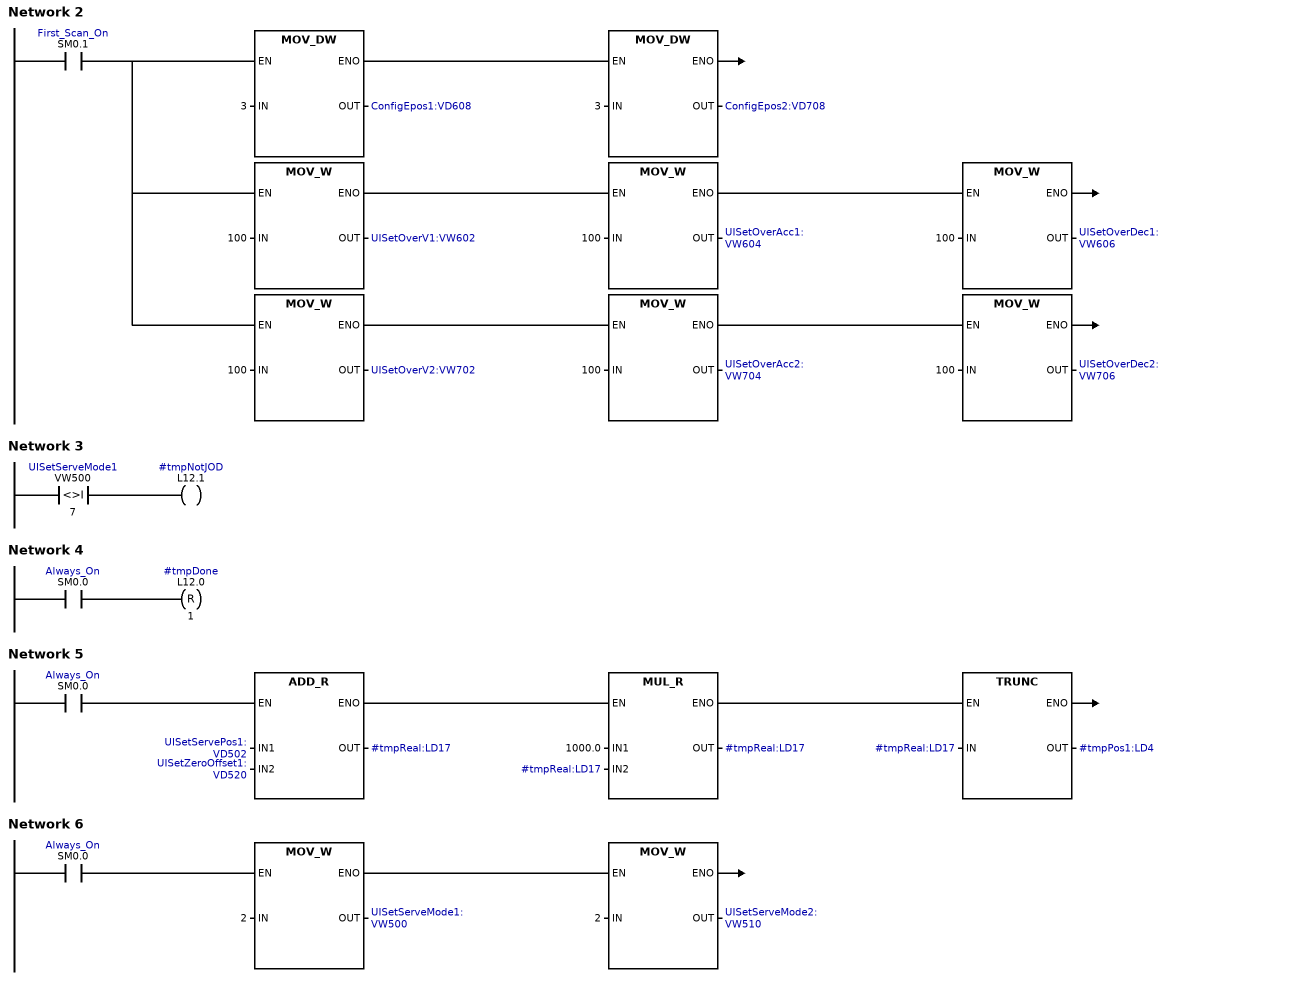
Network 2
LD     First_Scan_On:SM0.1
LPS
MOVD   3, ConfigEpos1:VD608
AENO
MOVD   3, ConfigEpos2:VD708
LRD
MOVW   100, UISetOverV1:VW602
AENO
MOVW   100, UISetOverAcc1:VW604
AENO
MOVW   100, UISetOverDec1:VW606
LPP
MOVW   100, UISetOverV2:VW702
AENO
MOVW   100, UISetOverAcc2:VW704
AENO
MOVW   100, UISetOverDec2:VW706
Network 3
LDW<>  UISetServeMode1:VW500, 7
=      #tmpNotJOD:L12.1
Network 4
LD     Always_On:SM0.0
R      #tmpDone:L12.0, 1
Network 5
LD     Always_On:SM0.0
MOVR   UISetServePos1:VD502, #tmpReal:LD17
AENO
+R     UISetZeroOffset1:VD520, #tmpReal:LD17
AENO
*R     1000.0, #tmpReal:LD17
AENO
TRUNC  #tmpReal:LD17, #tmpPos1:LD4
Network 6
LD     Always_On:SM0.0
MOVW   2, UISetServeMode1:VW500
AENO
MOVW   2, UISetServeMode2:VW510
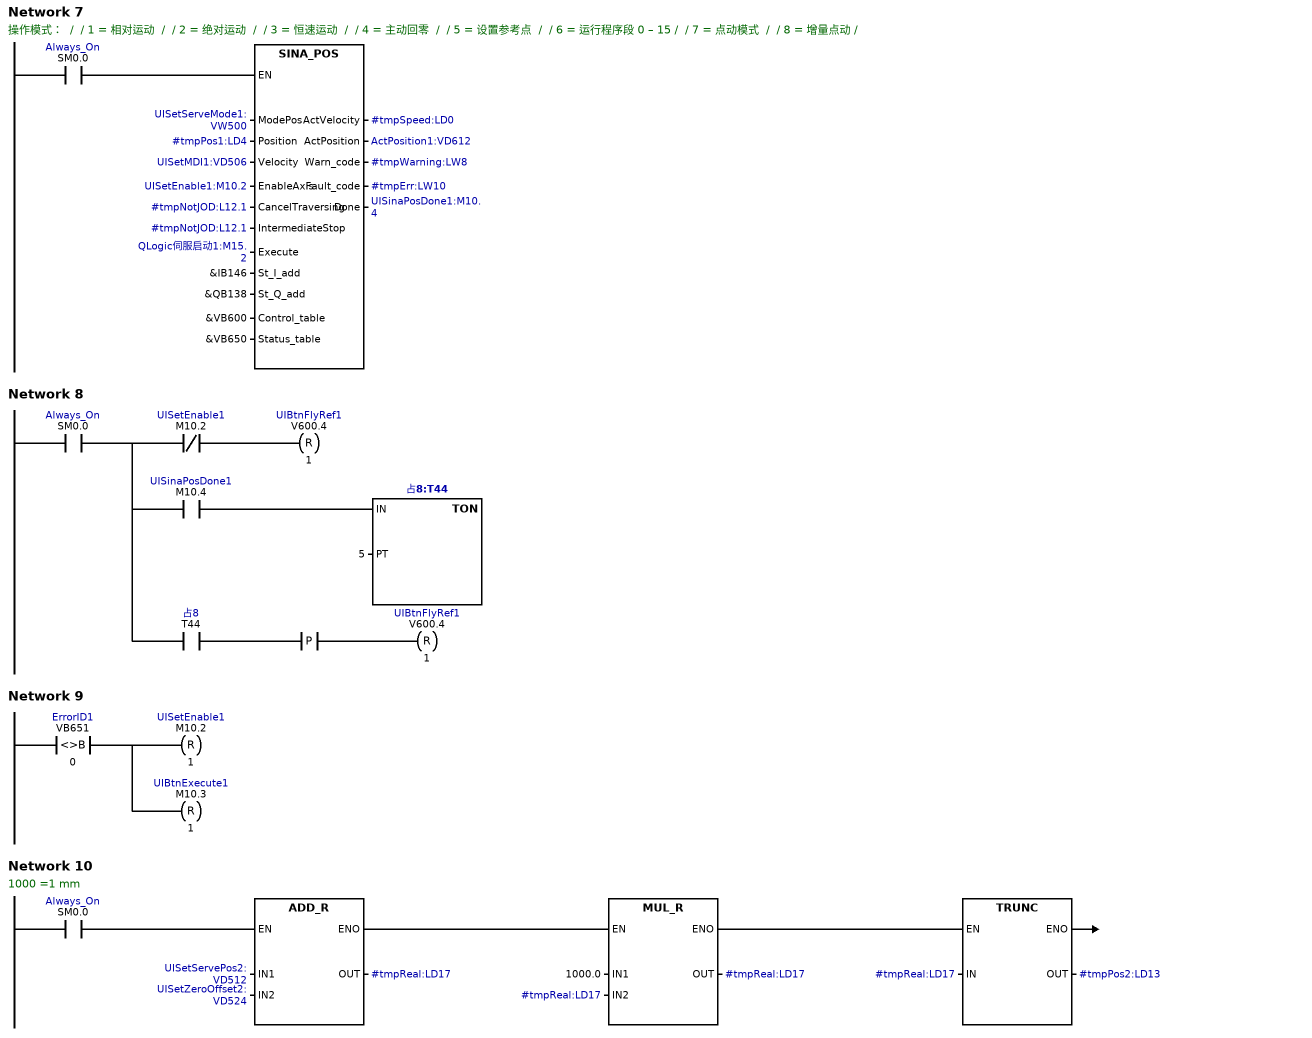
Network 7
// 操作模式： 
// 
// 1 = 相对运动 
// 
// 2 = 绝对运动 
// 
// 3 = 恒速运动 
// 
// 4 = 主动回零 
// 
// 5 = 设置参考点 
// 
// 6 = 运行程序段 0 – 15
// 
// 7 = 点动模式 
// 
// 8 = 增量点动
// 
LD     Always_On:SM0.0
CALL   SINA_POS:SBR8, UISetServeMode1:VW500, #tmpPos1:LD4, UISetMDI1:VD506, UISetEnable1:M10.2, #tmpNotJOD:L12.1, #tmpNotJOD:L12.1, QLogic伺服启动1:M15.2, &IB146, &QB138, &VB600, &VB650, #tmpSpeed:LD0, ActPosition1:VD612, #tmpWarning:LW8, #tmpErr:LW10, UISinaPosDone1:M10.4
Network 8
LD     Always_On:SM0.0
LPS
AN     UISetEnable1:M10.2
R      UIBtnFlyRef1:V600.4, 1
LRD
A      UISinaPosDone1:M10.4
TON    占8:T44, 5
LPP
A      占8:T44
EU
R      UIBtnFlyRef1:V600.4, 1
Network 9
LDB<>  ErrorID1:VB651, 0
R      UISetEnable1:M10.2, 1
R      UIBtnExecute1:M10.3, 1
Network 10
//  1000 =1 mm
LD     Always_On:SM0.0
MOVR   UISetServePos2:VD512, #tmpReal:LD17
AENO
+R     UISetZeroOffset2:VD524, #tmpReal:LD17
AENO
*R     1000.0, #tmpReal:LD17
AENO
TRUNC  #tmpReal:LD17, #tmpPos2:LD13
